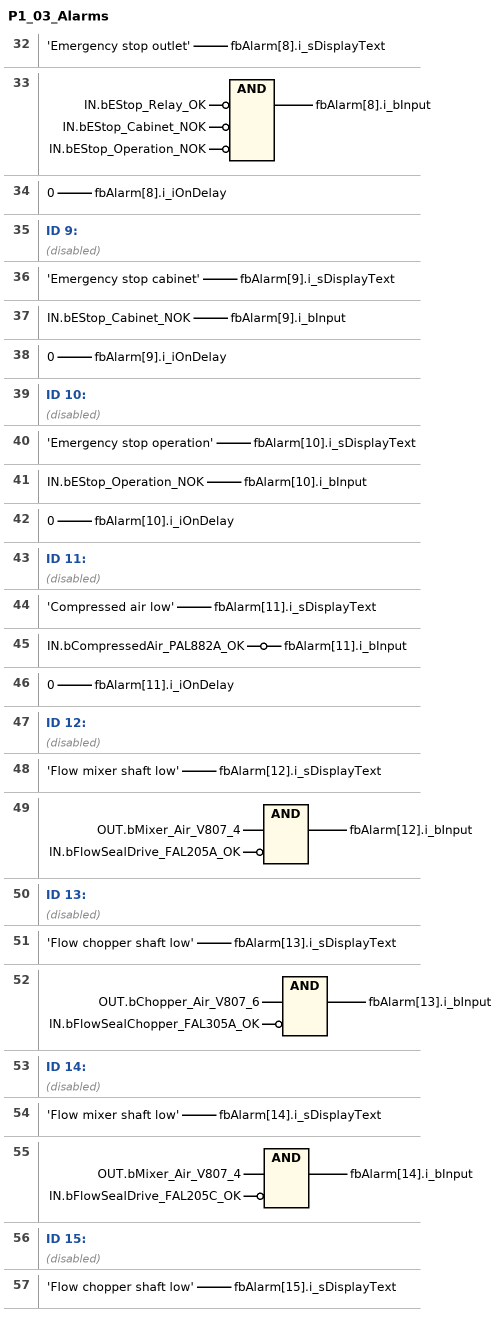
// NETWORK 32
fbAlarm[8].i_sDisplayText := 'Emergency stop outlet';

// NETWORK 33
fbAlarm[8].i_bInput := NOT IN.bEStop_Relay_OK AND NOT IN.bEStop_Cabinet_NOK AND NOT IN.bEStop_Operation_NOK;

// NETWORK 34
fbAlarm[8].i_iOnDelay := 0;

// NETWORK 35 (disabled)
// label: ID 9

// NETWORK 36
fbAlarm[9].i_sDisplayText := 'Emergency stop cabinet';

// NETWORK 37
fbAlarm[9].i_bInput := IN.bEStop_Cabinet_NOK;

// NETWORK 38
fbAlarm[9].i_iOnDelay := 0;

// NETWORK 39 (disabled)
// label: ID 10

// NETWORK 40
fbAlarm[10].i_sDisplayText := 'Emergency stop operation';

// NETWORK 41
fbAlarm[10].i_bInput := IN.bEStop_Operation_NOK;

// NETWORK 42
fbAlarm[10].i_iOnDelay := 0;

// NETWORK 43 (disabled)
// label: ID 11

// NETWORK 44
fbAlarm[11].i_sDisplayText := 'Compressed air low';

// NETWORK 45
fbAlarm[11].i_bInput := NOT IN.bCompressedAir_PAL882A_OK;

// NETWORK 46
fbAlarm[11].i_iOnDelay := 0;

// NETWORK 47 (disabled)
// label: ID 12

// NETWORK 48
fbAlarm[12].i_sDisplayText := 'Flow mixer shaft low';

// NETWORK 49
fbAlarm[12].i_bInput := OUT.bMixer_Air_V807_4 AND NOT IN.bFlowSealDrive_FAL205A_OK;

// NETWORK 50 (disabled)
// label: ID 13

// NETWORK 51
fbAlarm[13].i_sDisplayText := 'Flow chopper shaft low';

// NETWORK 52
fbAlarm[13].i_bInput := OUT.bChopper_Air_V807_6 AND NOT IN.bFlowSealChopper_FAL305A_OK;

// NETWORK 53 (disabled)
// label: ID 14

// NETWORK 54
fbAlarm[14].i_sDisplayText := 'Flow mixer shaft low';

// NETWORK 55
fbAlarm[14].i_bInput := OUT.bMixer_Air_V807_4 AND NOT IN.bFlowSealDrive_FAL205C_OK;

// NETWORK 56 (disabled)
// label: ID 15

// NETWORK 57
fbAlarm[15].i_sDisplayText := 'Flow chopper shaft low';

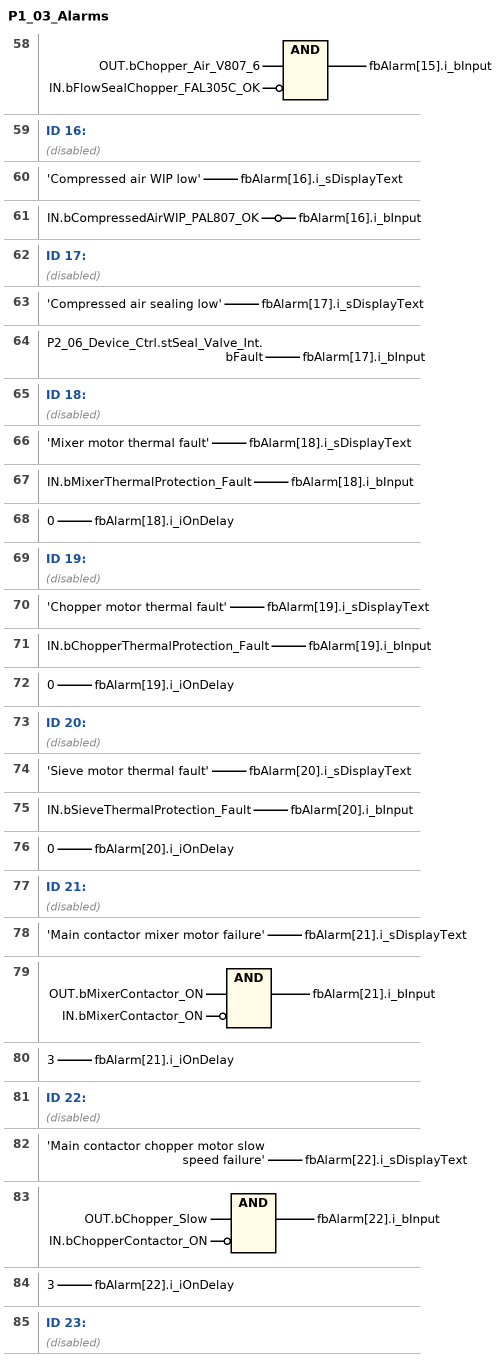
// NETWORK 58
fbAlarm[15].i_bInput := OUT.bChopper_Air_V807_6 AND NOT IN.bFlowSealChopper_FAL305C_OK;

// NETWORK 59 (disabled)
// label: ID 16

// NETWORK 60
fbAlarm[16].i_sDisplayText := 'Compressed air WIP low';

// NETWORK 61
fbAlarm[16].i_bInput := NOT IN.bCompressedAirWIP_PAL807_OK;

// NETWORK 62 (disabled)
// label: ID 17

// NETWORK 63
fbAlarm[17].i_sDisplayText := 'Compressed air sealing low';

// NETWORK 64
fbAlarm[17].i_bInput := P2_06_Device_Ctrl.stSeal_Valve_Int.bFault;

// NETWORK 65 (disabled)
// label: ID 18

// NETWORK 66
fbAlarm[18].i_sDisplayText := 'Mixer motor thermal fault';

// NETWORK 67
fbAlarm[18].i_bInput := IN.bMixerThermalProtection_Fault;

// NETWORK 68
fbAlarm[18].i_iOnDelay := 0;

// NETWORK 69 (disabled)
// label: ID 19

// NETWORK 70
fbAlarm[19].i_sDisplayText := 'Chopper motor thermal fault';

// NETWORK 71
fbAlarm[19].i_bInput := IN.bChopperThermalProtection_Fault;

// NETWORK 72
fbAlarm[19].i_iOnDelay := 0;

// NETWORK 73 (disabled)
// label: ID 20

// NETWORK 74
fbAlarm[20].i_sDisplayText := 'Sieve motor thermal fault';

// NETWORK 75
fbAlarm[20].i_bInput := IN.bSieveThermalProtection_Fault;

// NETWORK 76
fbAlarm[20].i_iOnDelay := 0;

// NETWORK 77 (disabled)
// label: ID 21

// NETWORK 78
fbAlarm[21].i_sDisplayText := 'Main contactor mixer motor failure';

// NETWORK 79
fbAlarm[21].i_bInput := OUT.bMixerContactor_ON AND NOT IN.bMixerContactor_ON;

// NETWORK 80
fbAlarm[21].i_iOnDelay := 3;

// NETWORK 81 (disabled)
// label: ID 22

// NETWORK 82
fbAlarm[22].i_sDisplayText := 'Main contactor chopper motor slow speed failure';

// NETWORK 83
fbAlarm[22].i_bInput := OUT.bChopper_Slow AND NOT IN.bChopperContactor_ON;

// NETWORK 84
fbAlarm[22].i_iOnDelay := 3;

// NETWORK 85 (disabled)
// label: ID 23

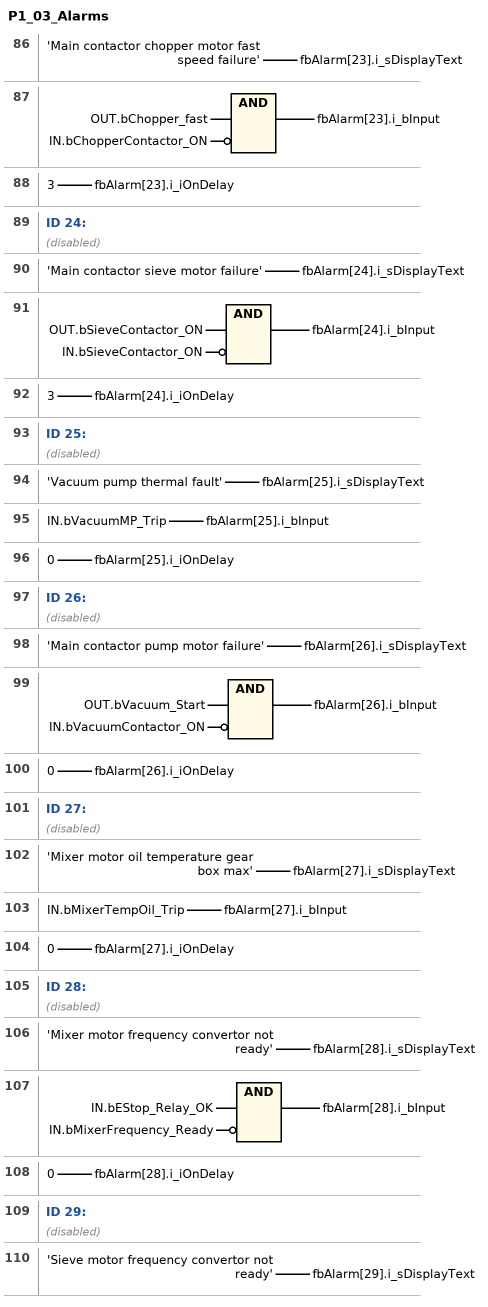
// NETWORK 86
fbAlarm[23].i_sDisplayText := 'Main contactor chopper motor fast speed failure';

// NETWORK 87
fbAlarm[23].i_bInput := OUT.bChopper_fast AND NOT IN.bChopperContactor_ON;

// NETWORK 88
fbAlarm[23].i_iOnDelay := 3;

// NETWORK 89 (disabled)
// label: ID 24

// NETWORK 90
fbAlarm[24].i_sDisplayText := 'Main contactor sieve motor failure';

// NETWORK 91
fbAlarm[24].i_bInput := OUT.bSieveContactor_ON AND NOT IN.bSieveContactor_ON;

// NETWORK 92
fbAlarm[24].i_iOnDelay := 3;

// NETWORK 93 (disabled)
// label: ID 25

// NETWORK 94
fbAlarm[25].i_sDisplayText := 'Vacuum pump thermal fault';

// NETWORK 95
fbAlarm[25].i_bInput := IN.bVacuumMP_Trip;

// NETWORK 96
fbAlarm[25].i_iOnDelay := 0;

// NETWORK 97 (disabled)
// label: ID 26

// NETWORK 98
fbAlarm[26].i_sDisplayText := 'Main contactor pump motor failure';

// NETWORK 99
fbAlarm[26].i_bInput := OUT.bVacuum_Start AND NOT IN.bVacuumContactor_ON;

// NETWORK 100
fbAlarm[26].i_iOnDelay := 0;

// NETWORK 101 (disabled)
// label: ID 27

// NETWORK 102
fbAlarm[27].i_sDisplayText := 'Mixer motor oil temperature gear box max';

// NETWORK 103
fbAlarm[27].i_bInput := IN.bMixerTempOil_Trip;

// NETWORK 104
fbAlarm[27].i_iOnDelay := 0;

// NETWORK 105 (disabled)
// label: ID 28

// NETWORK 106
fbAlarm[28].i_sDisplayText := 'Mixer motor frequency convertor not ready';

// NETWORK 107
fbAlarm[28].i_bInput := IN.bEStop_Relay_OK AND NOT IN.bMixerFrequency_Ready;

// NETWORK 108
fbAlarm[28].i_iOnDelay := 0;

// NETWORK 109 (disabled)
// label: ID 29

// NETWORK 110
fbAlarm[29].i_sDisplayText := 'Sieve motor frequency convertor not ready';

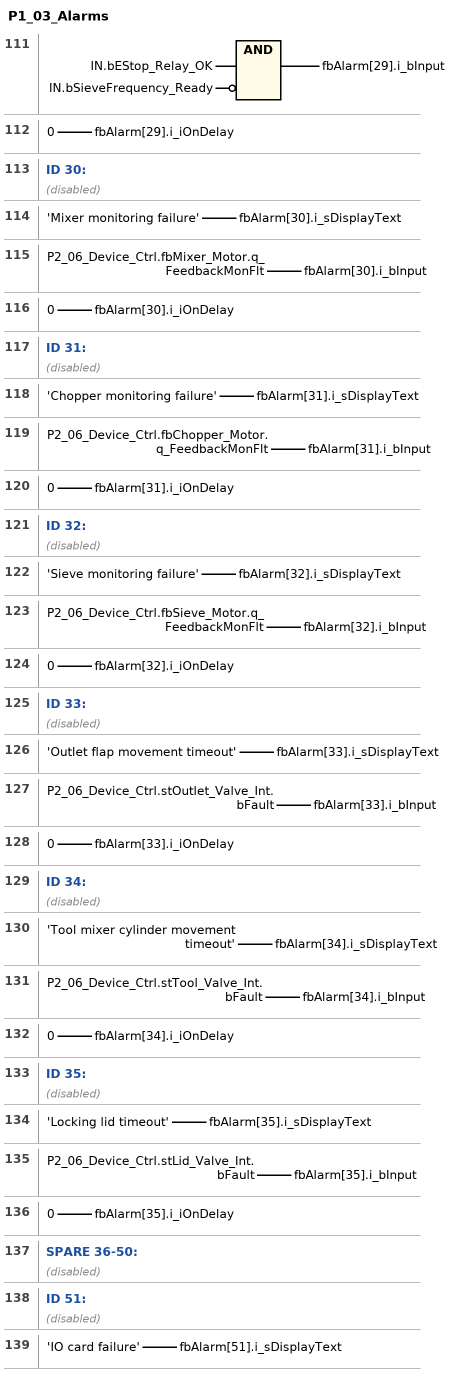
// NETWORK 111
fbAlarm[29].i_bInput := IN.bEStop_Relay_OK AND NOT IN.bSieveFrequency_Ready;

// NETWORK 112
fbAlarm[29].i_iOnDelay := 0;

// NETWORK 113 (disabled)
// label: ID 30

// NETWORK 114
fbAlarm[30].i_sDisplayText := 'Mixer monitoring failure';

// NETWORK 115
fbAlarm[30].i_bInput := P2_06_Device_Ctrl.fbMixer_Motor.q_FeedbackMonFlt;

// NETWORK 116
fbAlarm[30].i_iOnDelay := 0;

// NETWORK 117 (disabled)
// label: ID 31

// NETWORK 118
fbAlarm[31].i_sDisplayText := 'Chopper monitoring failure';

// NETWORK 119
fbAlarm[31].i_bInput := P2_06_Device_Ctrl.fbChopper_Motor.q_FeedbackMonFlt;

// NETWORK 120
fbAlarm[31].i_iOnDelay := 0;

// NETWORK 121 (disabled)
// label: ID 32

// NETWORK 122
fbAlarm[32].i_sDisplayText := 'Sieve monitoring failure';

// NETWORK 123
fbAlarm[32].i_bInput := P2_06_Device_Ctrl.fbSieve_Motor.q_FeedbackMonFlt;

// NETWORK 124
fbAlarm[32].i_iOnDelay := 0;

// NETWORK 125 (disabled)
// label: ID 33

// NETWORK 126
fbAlarm[33].i_sDisplayText := 'Outlet flap movement timeout';

// NETWORK 127
fbAlarm[33].i_bInput := P2_06_Device_Ctrl.stOutlet_Valve_Int.bFault;

// NETWORK 128
fbAlarm[33].i_iOnDelay := 0;

// NETWORK 129 (disabled)
// label: ID 34

// NETWORK 130
fbAlarm[34].i_sDisplayText := 'Tool mixer cylinder movement timeout';

// NETWORK 131
fbAlarm[34].i_bInput := P2_06_Device_Ctrl.stTool_Valve_Int.bFault;

// NETWORK 132
fbAlarm[34].i_iOnDelay := 0;

// NETWORK 133 (disabled)
// label: ID 35

// NETWORK 134
fbAlarm[35].i_sDisplayText := 'Locking lid timeout';

// NETWORK 135
fbAlarm[35].i_bInput := P2_06_Device_Ctrl.stLid_Valve_Int.bFault;

// NETWORK 136
fbAlarm[35].i_iOnDelay := 0;

// NETWORK 137 (disabled)
// label: SPARE 36-50

// NETWORK 138 (disabled)
// label: ID 51

// NETWORK 139
fbAlarm[51].i_sDisplayText := 'IO card failure';

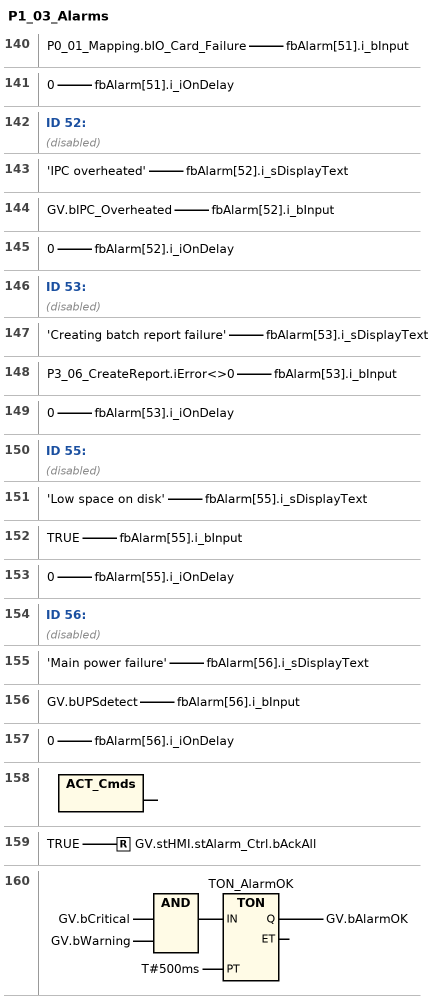
// NETWORK 140
fbAlarm[51].i_bInput := P0_01_Mapping.bIO_Card_Failure;

// NETWORK 141
fbAlarm[51].i_iOnDelay := 0;

// NETWORK 142 (disabled)
// label: ID 52

// NETWORK 143
fbAlarm[52].i_sDisplayText := 'IPC overheated';

// NETWORK 144
fbAlarm[52].i_bInput := GV.bIPC_Overheated;

// NETWORK 145
fbAlarm[52].i_iOnDelay := 0;

// NETWORK 146 (disabled)
// label: ID 53

// NETWORK 147
fbAlarm[53].i_sDisplayText := 'Creating batch report failure';

// NETWORK 148
fbAlarm[53].i_bInput := P3_06_CreateReport.iError<>0;

// NETWORK 149
fbAlarm[53].i_iOnDelay := 0;

// NETWORK 150 (disabled)
// label: ID 55

// NETWORK 151
fbAlarm[55].i_sDisplayText := 'Low space on disk';

// NETWORK 152
fbAlarm[55].i_bInput := TRUE;

// NETWORK 153
fbAlarm[55].i_iOnDelay := 0;

// NETWORK 154 (disabled)
// label: ID 56

// NETWORK 155
fbAlarm[56].i_sDisplayText := 'Main power failure';

// NETWORK 156
fbAlarm[56].i_bInput := GV.bUPSdetect;

// NETWORK 157
fbAlarm[56].i_iOnDelay := 0;

// NETWORK 158
ACT_Cmds();

// NETWORK 159
GV.stHMI.stAlarm_Ctrl.bAckAll R= TRUE;

// NETWORK 160
TON_AlarmOK(IN := GV.bCritical AND GV.bWarning, PT := T#500ms); // TON
GV.bAlarmOK := TON_AlarmOK.Q;

ACTION ACT_Cmds:
GV.bCritical:=TRUE;
GV.bWarning:=TRUE;
bAlarmDisabled:=FALSE;
FOR i:=0 TO 50 DO
	//Init Function blocks
	fbAlarm[i](i_iID:=i,
			   i_bActive:=GV.stAlarm.Active[i],
			   q_bActive=>GV.stAlarm.Raise[i]);			
			   
	fbAlarm[i].i_bEnable:=TRUE;
	IF GV.stAlarm.Active[i] THEN
		IF i <= 25 THEN
			GV.bCritical:=FALSE;
		ELSIF i > 25 THEN
			GV.bWarning:=FALSE;
		END_IF
	END_IF
	
	//Raise
	IF GV.stAlarm.Raise[i] THEN
		GV.stAlarm.Alarm[i].Raise(0);
	END_IF
	
	//Active
	GV.stAlarm.Active[i]:=GV.stAlarm.Alarm[i].bActive;
	
	//Ack
	IF GV.stAlarm.Alarm[i].eConfirmationState = 3 OR GV.stHMI.stAlarm_Ctrl.bAckAll THEN
		GV.stAlarm.Alarm[i].Clear(0,1);
	END_IF
	
	//Clear warnings 
	IF GV.stAlarm.Active[i] AND NOT fbAlarm[i].i_bInput AND i>=25 THEN
		GV.stAlarm.Alarm[i].Clear(0,1);
	END_IF
	
	//Check disabled
	IF NOT fbAlarm[i].i_bEnable THEN
		bAlarmDisabled:=TRUE;
	END_IF
END_FOR
END_ACTION

ACTION ACT_Init:
IF MAIN.bFirstCycle THEN
	//Critical
	GV.stAlarm.Alarm[1].CreateEx(TC_EVENTS.Alarms.AlarmsEvent1,1,0);
	GV.stAlarm.Alarm[2].CreateEx(TC_EVENTS.Alarms.AlarmsEvent2,1,0);
	GV.stAlarm.Alarm[3].CreateEx(TC_EVENTS.Alarms.AlarmsEvent3,1,0);
	GV.stAlarm.Alarm[4].CreateEx(TC_EVENTS.Alarms.AlarmsEvent4,1,0);
	GV.stAlarm.Alarm[5].CreateEx(TC_EVENTS.Alarms.AlarmsEvent5,1,0);
	GV.stAlarm.Alarm[6].CreateEx(TC_EVENTS.Alarms.AlarmsEvent6,1,0);
	GV.stAlarm.Alarm[7].CreateEx(TC_EVENTS.Alarms.AlarmsEvent7,1,0);
	GV.stAlarm.Alarm[8].CreateEx(TC_EVENTS.Alarms.AlarmsEvent8,1,0);
	GV.stAlarm.Alarm[9].CreateEx(TC_EVENTS.Alarms.AlarmsEvent9,1,0);
	GV.stAlarm.Alarm[10].CreateEx(TC_EVENTS.Alarms.AlarmsEvent10,1,0);
	GV.stAlarm.Alarm[11].CreateEx(TC_EVENTS.Alarms.AlarmsEvent11,1,0);
	GV.stAlarm.Alarm[12].CreateEx(TC_EVENTS.Alarms.AlarmsEvent12,1,0);
	GV.stAlarm.Alarm[13].CreateEx(TC_EVENTS.Alarms.AlarmsEvent13,1,0);
	GV.stAlarm.Alarm[14].CreateEx(TC_EVENTS.Alarms.AlarmsEvent14,1,0);
	GV.stAlarm.Alarm[15].CreateEx(TC_EVENTS.Alarms.AlarmsEvent15,1,0);
	GV.stAlarm.Alarm[16].CreateEx(TC_EVENTS.Alarms.AlarmsEvent16,1,0);
	GV.stAlarm.Alarm[17].CreateEx(TC_EVENTS.Alarms.AlarmsEvent17,1,0);
	GV.stAlarm.Alarm[18].CreateEx(TC_EVENTS.Alarms.AlarmsEvent18,1,0);
	GV.stAlarm.Alarm[19].CreateEx(TC_EVENTS.Alarms.AlarmsEvent19,1,0);
	GV.stAlarm.Alarm[20].CreateEx(TC_EVENTS.Alarms.AlarmsEvent20,1,0);
	GV.stAlarm.Alarm[21].CreateEx(TC_EVENTS.Alarms.AlarmsEvent21,1,0);
	GV.stAlarm.Alarm[22].CreateEx(TC_EVENTS.Alarms.AlarmsEvent22,1,0);
	GV.stAlarm.Alarm[23].CreateEx(TC_EVENTS.Alarms.AlarmsEvent23,1,0);
	GV.stAlarm.Alarm[24].CreateEx(TC_EVENTS.Alarms.AlarmsEvent24,1,0);
	GV.stAlarm.Alarm[25].CreateEx(TC_EVENTS.Alarms.AlarmsEvent25,1,0);
	GV.stAlarm.Alarm[26].CreateEx(TC_EVENTS.Alarms.AlarmsEvent26,1,0);
	GV.stAlarm.Alarm[27].CreateEx(TC_EVENTS.Alarms.AlarmsEvent27,1,0);
	GV.stAlarm.Alarm[28].CreateEx(TC_EVENTS.Alarms.AlarmsEvent28,1,0);
	GV.stAlarm.Alarm[29].CreateEx(TC_EVENTS.Alarms.AlarmsEvent29,1,0);
	GV.stAlarm.Alarm[30].CreateEx(TC_EVENTS.Alarms.AlarmsEvent30,1,0);
	GV.stAlarm.Alarm[31].CreateEx(TC_EVENTS.Alarms.AlarmsEvent31,1,0);
	GV.stAlarm.Alarm[32].CreateEx(TC_EVENTS.Alarms.AlarmsEvent32,1,0);
	GV.stAlarm.Alarm[33].CreateEx(TC_EVENTS.Alarms.AlarmsEvent33,1,0);
	GV.stAlarm.Alarm[34].CreateEx(TC_EVENTS.Alarms.AlarmsEvent34,1,0);
	GV.stAlarm.Alarm[35].CreateEx(TC_EVENTS.Alarms.AlarmsEvent35,1,0);
	GV.stAlarm.Alarm[36].CreateEx(TC_EVENTS.Alarms.AlarmsEvent36,1,0);
	GV.stAlarm.Alarm[37].CreateEx(TC_EVENTS.Alarms.AlarmsEvent37,1,0);
	GV.stAlarm.Alarm[38].CreateEx(TC_EVENTS.Alarms.AlarmsEvent38,1,0);
	GV.stAlarm.Alarm[39].CreateEx(TC_EVENTS.Alarms.AlarmsEvent39,1,0);
	GV.stAlarm.Alarm[40].CreateEx(TC_EVENTS.Alarms.AlarmsEvent40,1,0);	
	GV.stAlarm.Alarm[41].CreateEx(TC_EVENTS.Alarms.AlarmsEvent41,1,0);
	GV.stAlarm.Alarm[42].CreateEx(TC_EVENTS.Alarms.AlarmsEvent42,1,0);
	GV.stAlarm.Alarm[43].CreateEx(TC_EVENTS.Alarms.AlarmsEvent43,1,0);
	GV.stAlarm.Alarm[44].CreateEx(TC_EVENTS.Alarms.AlarmsEvent44,1,0);
	GV.stAlarm.Alarm[45].CreateEx(TC_EVENTS.Alarms.AlarmsEvent45,1,0);
	GV.stAlarm.Alarm[46].CreateEx(TC_EVENTS.Alarms.AlarmsEvent46,1,0);
	GV.stAlarm.Alarm[47].CreateEx(TC_EVENTS.Alarms.AlarmsEvent47,1,0);
	GV.stAlarm.Alarm[48].CreateEx(TC_EVENTS.Alarms.AlarmsEvent48,1,0);
	GV.stAlarm.Alarm[49].CreateEx(TC_EVENTS.Alarms.AlarmsEvent49,1,0);
	GV.stAlarm.Alarm[50].CreateEx(TC_EVENTS.Alarms.AlarmsEvent50,1,0);
	GV.stAlarm.Alarm[51].CreateEx(TC_EVENTS.Alarms.AlarmsEvent51,1,0);
	GV.stAlarm.Alarm[52].CreateEx(TC_EVENTS.Alarms.AlarmsEvent52,1,0);
	GV.stAlarm.Alarm[53].CreateEx(TC_EVENTS.Alarms.AlarmsEvent53,1,0);
	GV.stAlarm.Alarm[54].CreateEx(TC_EVENTS.Alarms.AlarmsEvent54,1,0);
	GV.stAlarm.Alarm[55].CreateEx(TC_EVENTS.Alarms.AlarmsEvent55,1,0);
	GV.stAlarm.Alarm[56].CreateEx(TC_EVENTS.Alarms.AlarmsEvent56,1,0);
	GV.stAlarm.Alarm[57].CreateEx(TC_EVENTS.Alarms.AlarmsEvent57,1,0);
	GV.stAlarm.Alarm[58].CreateEx(TC_EVENTS.Alarms.AlarmsEvent58,1,0);
	GV.stAlarm.Alarm[59].CreateEx(TC_EVENTS.Alarms.AlarmsEvent59,1,0);
	GV.stAlarm.Alarm[60].CreateEx(TC_EVENTS.Alarms.AlarmsEvent60,1,0);
	//SP
	GV.stAlarm.Alarm[61].CreateEx(TC_EVENTS.Alarms.AlarmsEvent61,1,0);
	GV.stAlarm.Alarm[62].CreateEx(TC_EVENTS.Alarms.AlarmsEvent62,1,0);
	GV.stAlarm.Alarm[63].CreateEx(TC_EVENTS.Alarms.AlarmsEvent63,1,0);
	GV.stAlarm.Alarm[64].CreateEx(TC_EVENTS.Alarms.AlarmsEvent64,1,0);
	GV.stAlarm.Alarm[65].CreateEx(TC_EVENTS.Alarms.AlarmsEvent65,1,0);
	GV.stAlarm.Alarm[66].CreateEx(TC_EVENTS.Alarms.AlarmsEvent66,1,0);
	GV.stAlarm.Alarm[67].CreateEx(TC_EVENTS.Alarms.AlarmsEvent67,1,0);
	GV.stAlarm.Alarm[68].CreateEx(TC_EVENTS.Alarms.AlarmsEvent68,1,0);
	GV.stAlarm.Alarm[69].CreateEx(TC_EVENTS.Alarms.AlarmsEvent69,1,0);
	GV.stAlarm.Alarm[70].CreateEx(TC_EVENTS.Alarms.AlarmsEvent70,1,0);
END_IF
END_ACTION

END_PROGRAM

// ---- FBs/FB_AlarmDiagnostic.TcPOU
FUNCTION_BLOCK FB_AlarmDiagnostic
VAR_INPUT
	i_bEnable				:BOOL:=TRUE;
	i_iID					:INT;
	i_bInput				:BOOL;
	i_iOnDelay				:INT;
	i_bReset				:BOOL;
	i_bTest					:BOOL;
	i_bActive				:BOOL;
END_VAR
VAR_OUTPUT
	q_bActive				:BOOL;
	q_iDetections			:INT;
END_VAR
VAR
	TON						:TON;
END_VAR
VAR // added by the converter: edge detectors and wires of the graphical bodies
    _rt1 : R_TRIG;
    _w1 : BOOL;
END_VAR

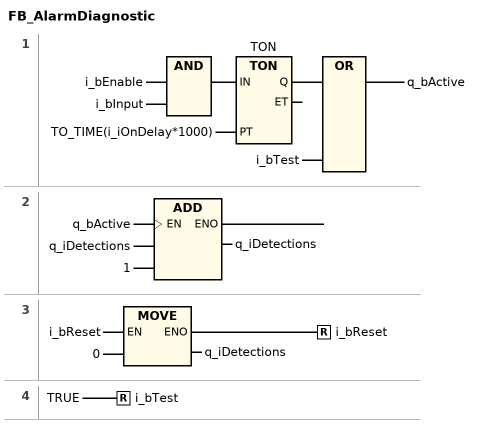
// NETWORK 1
TON(IN := i_bEnable AND i_bInput, PT := TO_TIME(i_iOnDelay*1000));
q_bActive := TON.Q OR i_bTest;

// NETWORK 2
_rt1(CLK := q_bActive);
IF _rt1.Q THEN q_iDetections := q_iDetections + 1; END_IF

// NETWORK 3
_w1 := i_bReset;
IF _w1 THEN q_iDetections := 0; END_IF
i_bReset R= _w1;

// NETWORK 4
i_bTest R= TRUE;

END_FUNCTION_BLOCK

// ---- POUs/2. Process/P2_06_Device_Ctrl.TcPOU
PROGRAM P2_06_Device_Ctrl
VAR
	fbMixer_Motor					:FB_MotorFreqCtrl;
	fbMixerMotor_Speed				:FB_AnalogOutput_v01;
	fbSieve_Motor					:FB_MotorFreqCtrl;
	fbSieveMotor_Speed				:FB_AnalogOutput_v01;
	fbChopper_Motor					:FB_MotorCoilsCtrl;
	fbPump_Motor					:FB_CoilCtrl;
	
	fbSP_Temperature_PID			:FB_PID;
	
	fbSP_Mixer_Motor				:FB_MotorFreqCtrl;
	fbSP_MixerMotor_Speed			:FB_AnalogOutput_v01;
	fbSP_Pressure					:FB_AnalogOutput_v02;
	
	fbOutlet_Valve					:FB_ValveCtrl52;
	fbLid_Valve						:FB_ValveCtrl52;
	fbSieveSeal_Valve				:FB_ValveCtrl52;
	fbPurge_Valve					:FB_ValveCtrl52;
	fbTool_Valve					:FB_ValveCtrl52;
	
	fbCleaningAir_Valve				:FB_ValveCtrl32;
	fbPurifiedWater_Valve			:FB_ValveCtrl32;
	fbWarmWater_Valve				:FB_ValveCtrl32;
	fbColdWater_Valve				:FB_ValveCtrl32;
	fbMixerWIP_Valve				:FB_ValveCtrl32;
	fbChopperWIP_Valve				:FB_ValveCtrl32;
	fbSPWIP_Valve					:FB_ValveCtrl32;
	fbSPWIPDrain_Valve				:FB_ValveCtrl32;
	fbMainDrain_Valve				:FB_ValveCtrl32;
	
	fbAspiration_Valve				:FB_ValveCtrl32;
	fbVacuum_Valve					:FB_ValveCtrl32;
	fbFilterClean_Valve				:FB_ValveCtrl32;
	fbAirSeal_Valve					:FB_ValveCtrl32;
	fbMixerAir_Valve				:FB_ValveCtrl32;
	fbChopperAir_Valve				:FB_ValveCtrl32;
	
	
	
	

END_VAR

VAR PERSISTENT
	stMixer_Motor_Int				:ST_Interface_MotorCtrl;
	stSieve_Motor_Int				:ST_Interface_MotorCtrl;
	stChopper_Motor_Int				:ST_Interface_MotorCoilsCtrl;
	stPump_Motor_Int				:ST_Interface_CoilCtrl;
	
	stSP_Mixer_Motor_Int			:ST_Interface_MotorCtrl;
	stSP_Temperature_Int			:ST_Interface_PidCtrl;
	
	stOutlet_Valve_Int				:ST_Interface_ValveCtrl;
	stLid_Valve_Int					:ST_Interface_ValveCtrl;
	stSeal_Valve_Int				:ST_Interface_ValveCtrl;
	stPurge_Valve_Int				:ST_Interface_ValveCtrl;
	stTool_Valve_Int				:ST_Interface_ValveCtrl;
	
	stCleaningAir_Valve_INT			:ST_Interface_ValveCtrl;
	stPurifiedWater_Valve_INT		:ST_Interface_ValveCtrl;
	stWarmWater_Valve_Int			:ST_Interface_ValveCtrl;
	stColdWater_Valve_Int			:ST_Interface_ValveCtrl;
	stMixerWIP_Valve_Int			:ST_Interface_ValveCtrl;
	stChopperWIP_Valve_Int			:ST_Interface_ValveCtrl;
	stSPWIP_Valve_Int				:ST_Interface_ValveCtrl;
	stSPWIPDrain_Valve_Int			:ST_Interface_ValveCtrl;
	stMainDrain_Valve_Int			:ST_Interface_ValveCtrl;
	
	stAspiration_Valve_Int			:ST_Interface_ValveCtrl;
	stVacuum_Valve_Int				:ST_Interface_ValveCtrl;
	stFilterClean_Valve_Int			:ST_Interface_ValveCtrl;
	stAirSeal_Valve_Int				:ST_Interface_ValveCtrl;
	stMixerAir_Valve_Int			:ST_Interface_ValveCtrl;
	stChopperAir_Valve_Int			:ST_Interface_ValveCtrl;
END_VAR
VAR // added by the converter: edge detectors and wires of the graphical bodies
    _w1, _w2, _w3, _w4, _w5, _w6, _w7, _w8, _w9, _w10 : BOOL;
    _rt1, _rt2 : R_TRIG;
END_VAR

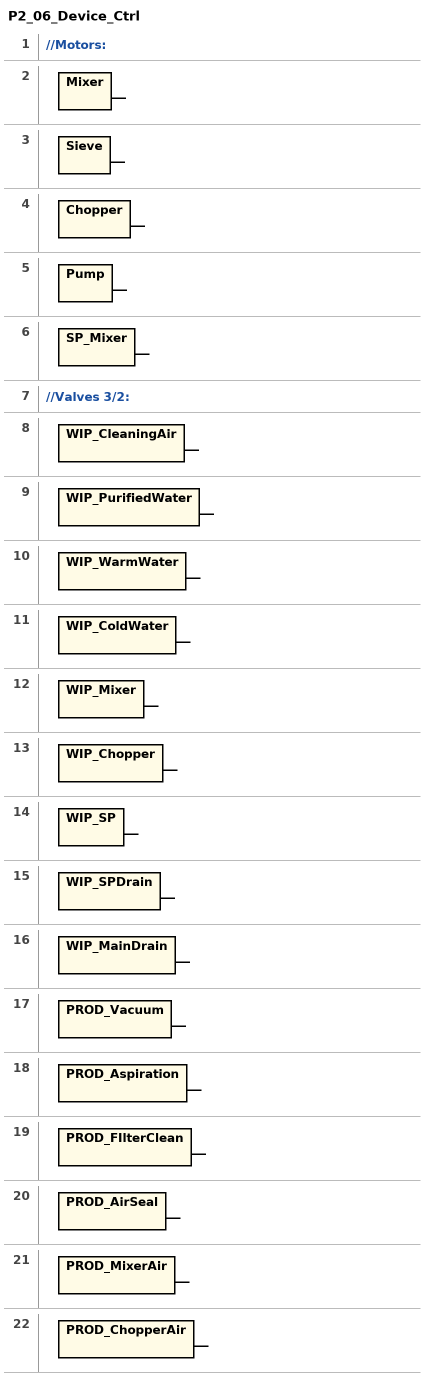
// NETWORK 1
// label: //Motors

// NETWORK 2
Mixer();

// NETWORK 3
Sieve();

// NETWORK 4
Chopper();

// NETWORK 5
Pump();

// NETWORK 6
SP_Mixer();

// NETWORK 7
// label: //Valves 3/2

// NETWORK 8
WIP_CleaningAir();

// NETWORK 9
WIP_PurifiedWater();

// NETWORK 10
WIP_WarmWater();

// NETWORK 11
WIP_ColdWater();

// NETWORK 12
WIP_Mixer();

// NETWORK 13
WIP_Chopper();

// NETWORK 14
WIP_SP();

// NETWORK 15
WIP_SPDrain();

// NETWORK 16
WIP_MainDrain();

// NETWORK 17
PROD_Vacuum();

// NETWORK 18
PROD_Aspiration();

// NETWORK 19
PROD_FIlterClean();

// NETWORK 20
PROD_AirSeal();

// NETWORK 21
PROD_MixerAir();

// NETWORK 22
PROD_ChopperAir();

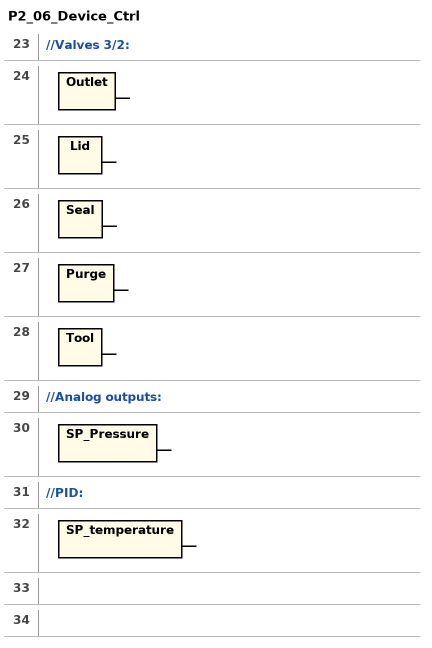
// NETWORK 23
// label: //Valves 3/2

// NETWORK 24
Outlet();

// NETWORK 25
Lid();

// NETWORK 26
Seal();

// NETWORK 27
Purge();

// NETWORK 28
Tool();

// NETWORK 29
// label: //Analog outputs

// NETWORK 30
SP_Pressure();

// NETWORK 31
// label: //PID

// NETWORK 32
SP_temperature();

// NETWORK 33

// NETWORK 34

ACTION Chopper:
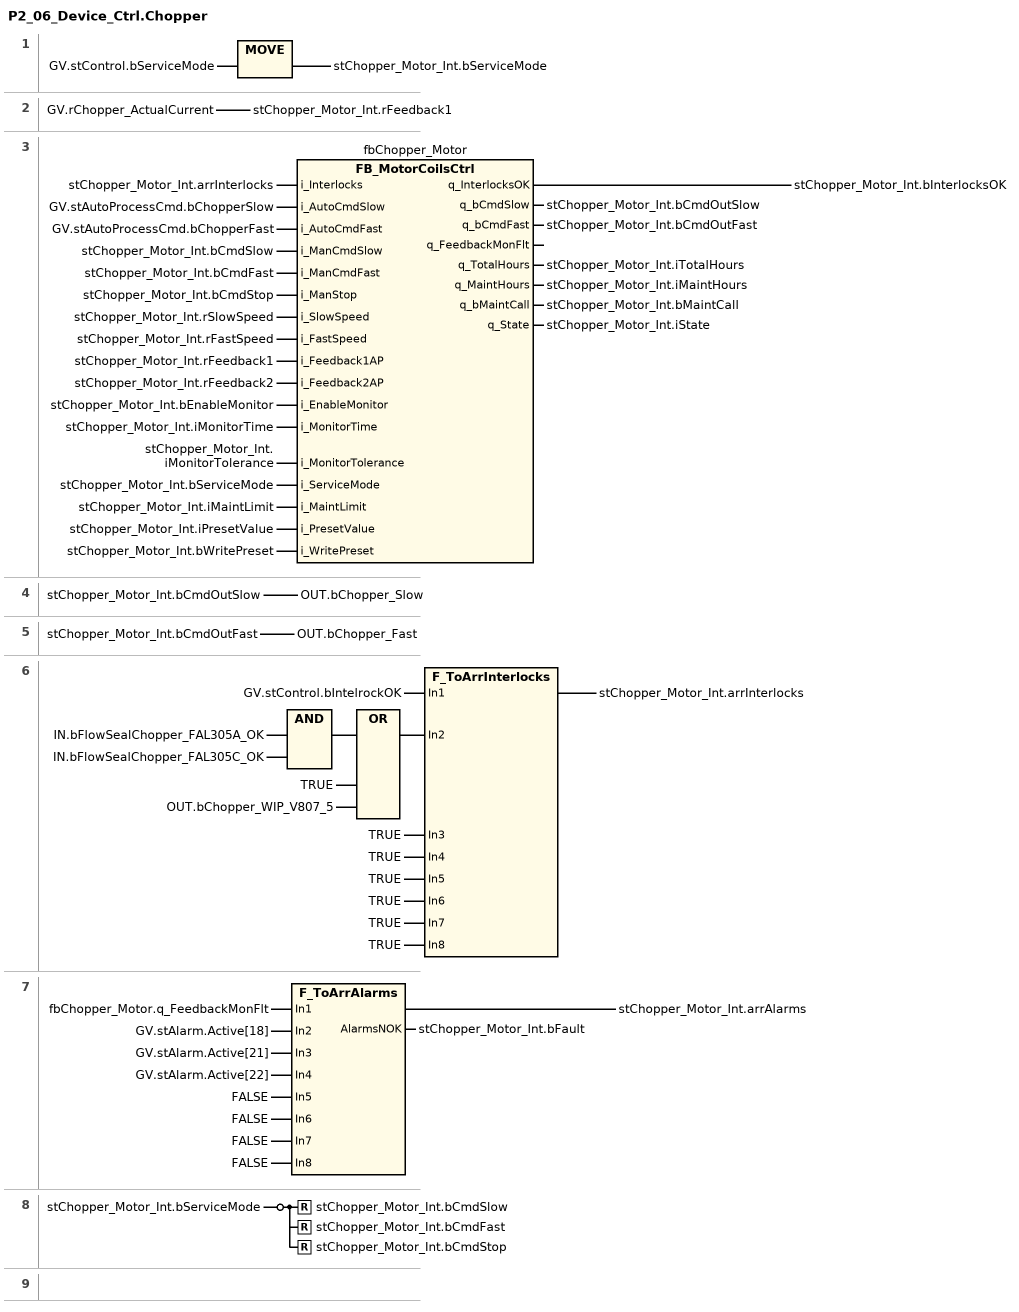
// NETWORK 1
stChopper_Motor_Int.bServiceMode := GV.stControl.bServiceMode;

// NETWORK 2
stChopper_Motor_Int.rFeedback1 := GV.rChopper_ActualCurrent;

// NETWORK 3
fbChopper_Motor(
    i_Interlocks := stChopper_Motor_Int.arrInterlocks,
    i_AutoCmdSlow := GV.stAutoProcessCmd.bChopperSlow,
    i_AutoCmdFast := GV.stAutoProcessCmd.bChopperFast,
    i_ManCmdSlow := stChopper_Motor_Int.bCmdSlow,
    i_ManCmdFast := stChopper_Motor_Int.bCmdFast,
    i_ManStop := stChopper_Motor_Int.bCmdStop,
    i_SlowSpeed := stChopper_Motor_Int.rSlowSpeed,
    i_FastSpeed := stChopper_Motor_Int.rFastSpeed,
    i_Feedback1AP := stChopper_Motor_Int.rFeedback1,
    i_Feedback2AP := stChopper_Motor_Int.rFeedback2,
    i_EnableMonitor := stChopper_Motor_Int.bEnableMonitor,
    i_MonitorTime := stChopper_Motor_Int.iMonitorTime,
    i_MonitorTolerance := stChopper_Motor_Int.iMonitorTolerance,
    i_ServiceMode := stChopper_Motor_Int.bServiceMode,
    i_MaintLimit := stChopper_Motor_Int.iMaintLimit,
    i_PresetValue := stChopper_Motor_Int.iPresetValue,
    i_WritePreset := stChopper_Motor_Int.bWritePreset,
    q_bCmdSlow => stChopper_Motor_Int.bCmdOutSlow,
    q_bCmdFast => stChopper_Motor_Int.bCmdOutFast,
    q_TotalHours => stChopper_Motor_Int.iTotalHours,
    q_MaintHours => stChopper_Motor_Int.iMaintHours,
    q_bMaintCall => stChopper_Motor_Int.bMaintCall,
    q_State => stChopper_Motor_Int.iState); // FB_MotorCoilsCtrl
stChopper_Motor_Int.bInterlocksOK := fbChopper_Motor.q_InterlocksOK;

// NETWORK 4
OUT.bChopper_Slow := stChopper_Motor_Int.bCmdOutSlow;

// NETWORK 5
OUT.bChopper_Fast := stChopper_Motor_Int.bCmdOutFast;

// NETWORK 6
stChopper_Motor_Int.arrInterlocks := F_ToArrInterlocks(In1 := GV.stControl.bIntelrockOK, In2 := IN.bFlowSealChopper_FAL305A_OK AND IN.bFlowSealChopper_FAL305C_OK OR TRUE OR OUT.bChopper_WIP_V807_5, In3 := TRUE, In4 := TRUE, In5 := TRUE, In6 := TRUE, In7 := TRUE, In8 := TRUE);

// NETWORK 7
stChopper_Motor_Int.arrAlarms := F_ToArrAlarms(In1 := fbChopper_Motor.q_FeedbackMonFlt, In2 := GV.stAlarm.Active[18], In3 := GV.stAlarm.Active[21], In4 := GV.stAlarm.Active[22], In5 := FALSE, In6 := FALSE, In7 := FALSE, In8 := FALSE, AlarmsNOK => stChopper_Motor_Int.bFault);

// NETWORK 8
_w1 := NOT stChopper_Motor_Int.bServiceMode;
stChopper_Motor_Int.bCmdSlow R= _w1;
stChopper_Motor_Int.bCmdFast R= _w1;
stChopper_Motor_Int.bCmdStop R= _w1;

// NETWORK 9
END_ACTION

ACTION Lid:
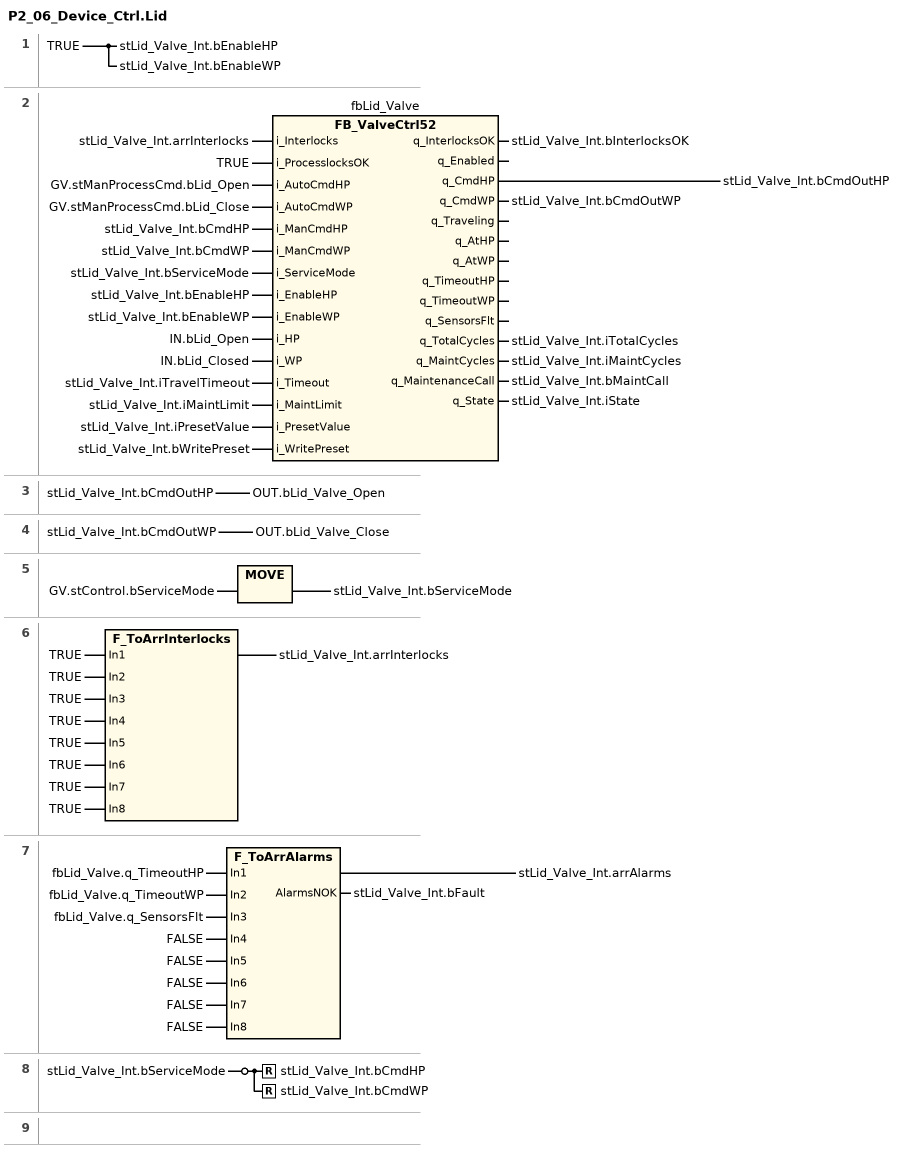
// NETWORK 1
stLid_Valve_Int.bEnableHP := TRUE;
stLid_Valve_Int.bEnableWP := TRUE;

// NETWORK 2
fbLid_Valve(
    i_Interlocks := stLid_Valve_Int.arrInterlocks,
    i_ProcesslocksOK := TRUE,
    i_AutoCmdHP := GV.stManProcessCmd.bLid_Open,
    i_AutoCmdWP := GV.stManProcessCmd.bLid_Close,
    i_ManCmdHP := stLid_Valve_Int.bCmdHP,
    i_ManCmdWP := stLid_Valve_Int.bCmdWP,
    i_ServiceMode := stLid_Valve_Int.bServiceMode,
    i_EnableHP := stLid_Valve_Int.bEnableHP,
    i_EnableWP := stLid_Valve_Int.bEnableWP,
    i_HP := IN.bLid_Open,
    i_WP := IN.bLid_Closed,
    i_Timeout := stLid_Valve_Int.iTravelTimeout,
    i_MaintLimit := stLid_Valve_Int.iMaintLimit,
    i_PresetValue := stLid_Valve_Int.iPresetValue,
    i_WritePreset := stLid_Valve_Int.bWritePreset,
    q_InterlocksOK => stLid_Valve_Int.bInterlocksOK,
    q_CmdWP => stLid_Valve_Int.bCmdOutWP,
    q_TotalCycles => stLid_Valve_Int.iTotalCycles,
    q_MaintCycles => stLid_Valve_Int.iMaintCycles,
    q_MaintenanceCall => stLid_Valve_Int.bMaintCall,
    q_State => stLid_Valve_Int.iState); // FB_ValveCtrl52
stLid_Valve_Int.bCmdOutHP := fbLid_Valve.q_CmdHP;

// NETWORK 3
OUT.bLid_Valve_Open := stLid_Valve_Int.bCmdOutHP;

// NETWORK 4
OUT.bLid_Valve_Close := stLid_Valve_Int.bCmdOutWP;

// NETWORK 5
stLid_Valve_Int.bServiceMode := GV.stControl.bServiceMode;

// NETWORK 6
stLid_Valve_Int.arrInterlocks := F_ToArrInterlocks(In1 := TRUE, In2 := TRUE, In3 := TRUE, In4 := TRUE, In5 := TRUE, In6 := TRUE, In7 := TRUE, In8 := TRUE);

// NETWORK 7
stLid_Valve_Int.arrAlarms := F_ToArrAlarms(In1 := fbLid_Valve.q_TimeoutHP, In2 := fbLid_Valve.q_TimeoutWP, In3 := fbLid_Valve.q_SensorsFlt, In4 := FALSE, In5 := FALSE, In6 := FALSE, In7 := FALSE, In8 := FALSE, AlarmsNOK => stLid_Valve_Int.bFault);

// NETWORK 8
_w2 := NOT stLid_Valve_Int.bServiceMode;
stLid_Valve_Int.bCmdHP R= _w2;
stLid_Valve_Int.bCmdWP R= _w2;

// NETWORK 9
END_ACTION

ACTION Mixer:
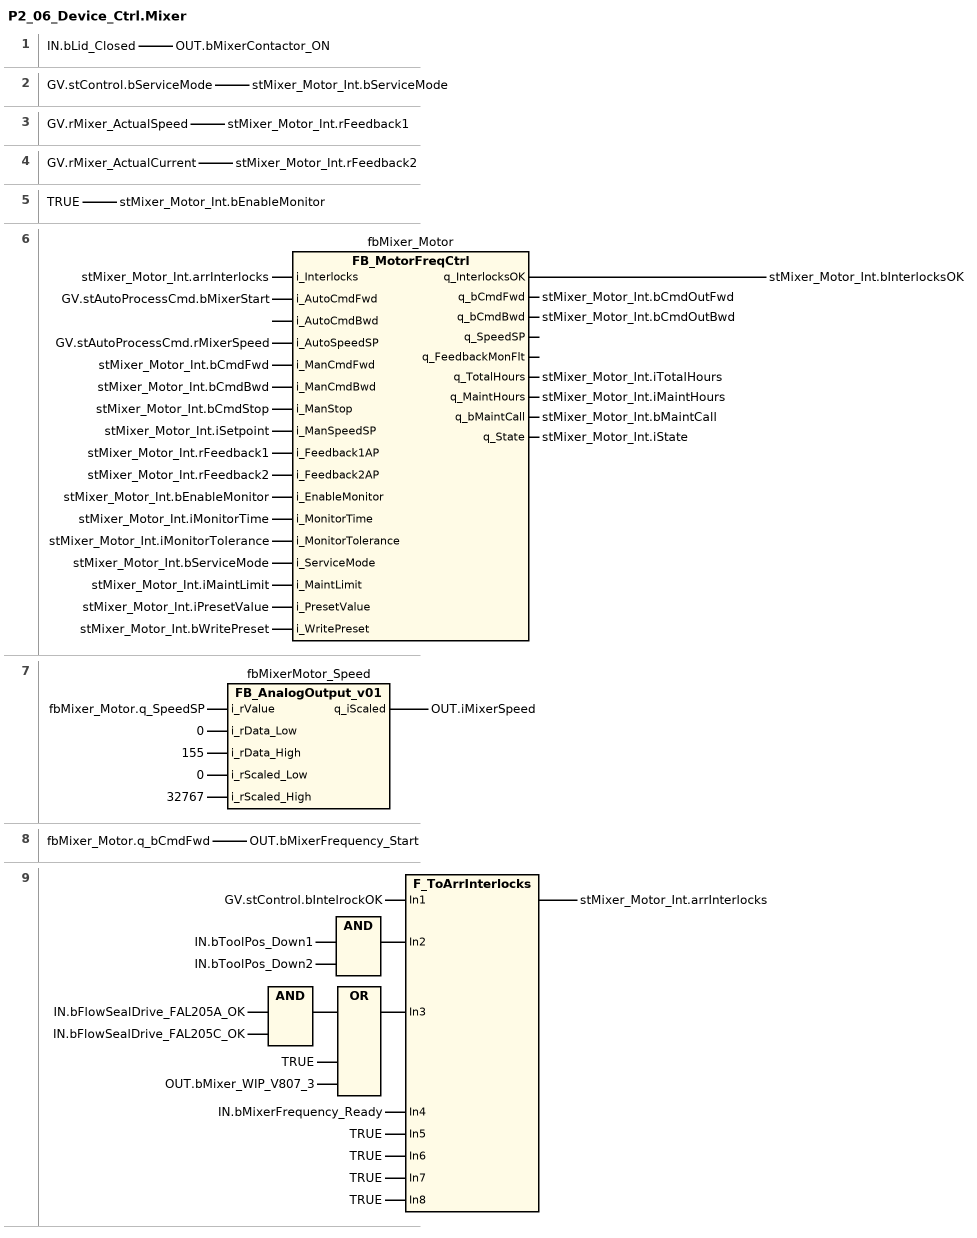
// NETWORK 1
OUT.bMixerContactor_ON := IN.bLid_Closed;

// NETWORK 2
stMixer_Motor_Int.bServiceMode := GV.stControl.bServiceMode;

// NETWORK 3
stMixer_Motor_Int.rFeedback1 := GV.rMixer_ActualSpeed;

// NETWORK 4
stMixer_Motor_Int.rFeedback2 := GV.rMixer_ActualCurrent;

// NETWORK 5
stMixer_Motor_Int.bEnableMonitor := TRUE;

// NETWORK 6
fbMixer_Motor(
    i_Interlocks := stMixer_Motor_Int.arrInterlocks,
    i_AutoCmdFwd := GV.stAutoProcessCmd.bMixerStart,
    i_AutoSpeedSP := GV.stAutoProcessCmd.rMixerSpeed,
    i_ManCmdFwd := stMixer_Motor_Int.bCmdFwd,
    i_ManCmdBwd := stMixer_Motor_Int.bCmdBwd,
    i_ManStop := stMixer_Motor_Int.bCmdStop,
    i_ManSpeedSP := stMixer_Motor_Int.iSetpoint,
    i_Feedback1AP := stMixer_Motor_Int.rFeedback1,
    i_Feedback2AP := stMixer_Motor_Int.rFeedback2,
    i_EnableMonitor := stMixer_Motor_Int.bEnableMonitor,
    i_MonitorTime := stMixer_Motor_Int.iMonitorTime,
    i_MonitorTolerance := stMixer_Motor_Int.iMonitorTolerance,
    i_ServiceMode := stMixer_Motor_Int.bServiceMode,
    i_MaintLimit := stMixer_Motor_Int.iMaintLimit,
    i_PresetValue := stMixer_Motor_Int.iPresetValue,
    i_WritePreset := stMixer_Motor_Int.bWritePreset,
    q_bCmdFwd => stMixer_Motor_Int.bCmdOutFwd,
    q_bCmdBwd => stMixer_Motor_Int.bCmdOutBwd,
    q_TotalHours => stMixer_Motor_Int.iTotalHours,
    q_MaintHours => stMixer_Motor_Int.iMaintHours,
    q_bMaintCall => stMixer_Motor_Int.bMaintCall,
    q_State => stMixer_Motor_Int.iState); // FB_MotorFreqCtrl
stMixer_Motor_Int.bInterlocksOK := fbMixer_Motor.q_InterlocksOK;

// NETWORK 7
fbMixerMotor_Speed(
    i_rValue := fbMixer_Motor.q_SpeedSP,
    i_rData_Low := 0,
    i_rData_High := 155,
    i_rScaled_Low := 0,
    i_rScaled_High := 32767); // FB_AnalogOutput_v01
OUT.iMixerSpeed := fbMixerMotor_Speed.q_iScaled;

// NETWORK 8
OUT.bMixerFrequency_Start := fbMixer_Motor.q_bCmdFwd;

// NETWORK 9
stMixer_Motor_Int.arrInterlocks := F_ToArrInterlocks(In1 := GV.stControl.bIntelrockOK, In2 := IN.bToolPos_Down1 AND IN.bToolPos_Down2, In3 := IN.bFlowSealDrive_FAL205A_OK AND IN.bFlowSealDrive_FAL205C_OK OR TRUE OR OUT.bMixer_WIP_V807_3, In4 := IN.bMixerFrequency_Ready, In5 := TRUE, In6 := TRUE, In7 := TRUE, In8 := TRUE);

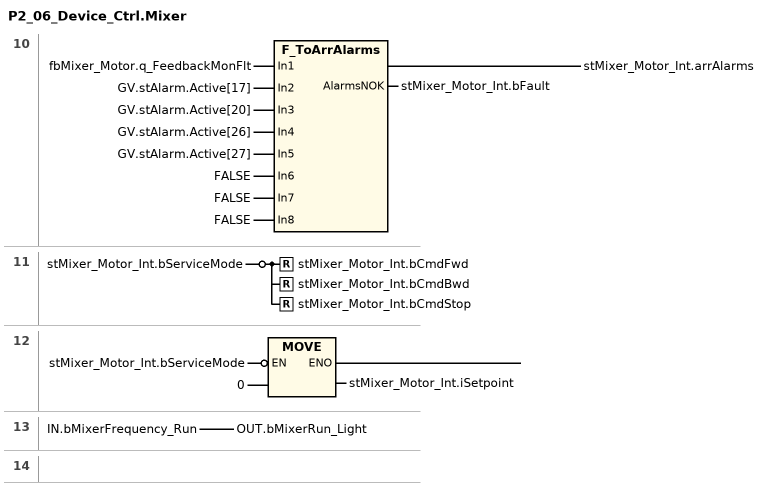
// NETWORK 10
stMixer_Motor_Int.arrAlarms := F_ToArrAlarms(In1 := fbMixer_Motor.q_FeedbackMonFlt, In2 := GV.stAlarm.Active[17], In3 := GV.stAlarm.Active[20], In4 := GV.stAlarm.Active[26], In5 := GV.stAlarm.Active[27], In6 := FALSE, In7 := FALSE, In8 := FALSE, AlarmsNOK => stMixer_Motor_Int.bFault);

// NETWORK 11
_w3 := NOT stMixer_Motor_Int.bServiceMode;
stMixer_Motor_Int.bCmdFwd R= _w3;
stMixer_Motor_Int.bCmdBwd R= _w3;
stMixer_Motor_Int.bCmdStop R= _w3;

// NETWORK 12
IF NOT stMixer_Motor_Int.bServiceMode THEN stMixer_Motor_Int.iSetpoint := 0; END_IF

// NETWORK 13
OUT.bMixerRun_Light := IN.bMixerFrequency_Run;

// NETWORK 14
END_ACTION

ACTION Outlet:
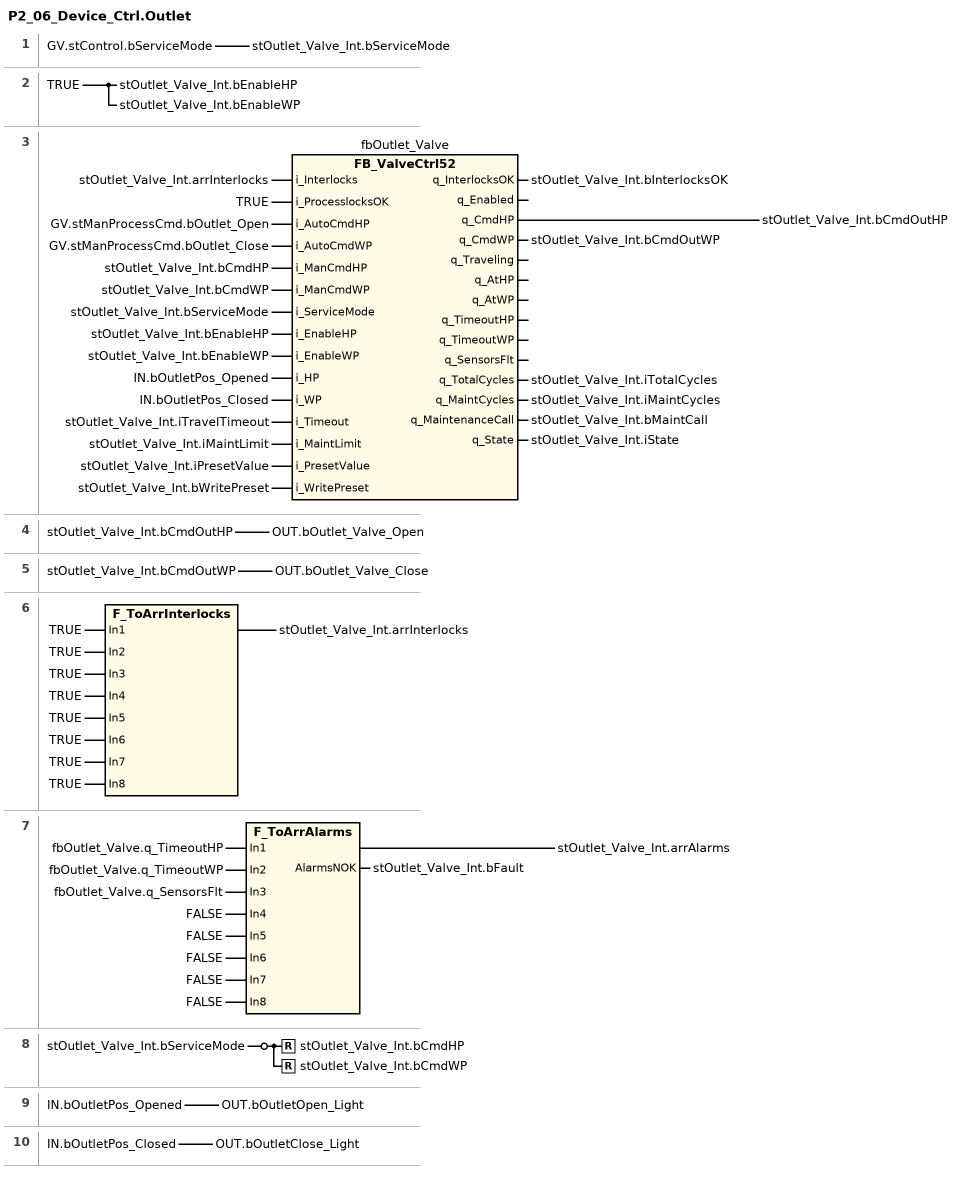
// NETWORK 1
stOutlet_Valve_Int.bServiceMode := GV.stControl.bServiceMode;

// NETWORK 2
stOutlet_Valve_Int.bEnableHP := TRUE;
stOutlet_Valve_Int.bEnableWP := TRUE;

// NETWORK 3
fbOutlet_Valve(
    i_Interlocks := stOutlet_Valve_Int.arrInterlocks,
    i_ProcesslocksOK := TRUE,
    i_AutoCmdHP := GV.stManProcessCmd.bOutlet_Open,
    i_AutoCmdWP := GV.stManProcessCmd.bOutlet_Close,
    i_ManCmdHP := stOutlet_Valve_Int.bCmdHP,
    i_ManCmdWP := stOutlet_Valve_Int.bCmdWP,
    i_ServiceMode := stOutlet_Valve_Int.bServiceMode,
    i_EnableHP := stOutlet_Valve_Int.bEnableHP,
    i_EnableWP := stOutlet_Valve_Int.bEnableWP,
    i_HP := IN.bOutletPos_Opened,
    i_WP := IN.bOutletPos_Closed,
    i_Timeout := stOutlet_Valve_Int.iTravelTimeout,
    i_MaintLimit := stOutlet_Valve_Int.iMaintLimit,
    i_PresetValue := stOutlet_Valve_Int.iPresetValue,
    i_WritePreset := stOutlet_Valve_Int.bWritePreset,
    q_InterlocksOK => stOutlet_Valve_Int.bInterlocksOK,
    q_CmdWP => stOutlet_Valve_Int.bCmdOutWP,
    q_TotalCycles => stOutlet_Valve_Int.iTotalCycles,
    q_MaintCycles => stOutlet_Valve_Int.iMaintCycles,
    q_MaintenanceCall => stOutlet_Valve_Int.bMaintCall,
    q_State => stOutlet_Valve_Int.iState); // FB_ValveCtrl52
stOutlet_Valve_Int.bCmdOutHP := fbOutlet_Valve.q_CmdHP;

// NETWORK 4
OUT.bOutlet_Valve_Open := stOutlet_Valve_Int.bCmdOutHP;

// NETWORK 5
OUT.bOutlet_Valve_Close := stOutlet_Valve_Int.bCmdOutWP;

// NETWORK 6
stOutlet_Valve_Int.arrInterlocks := F_ToArrInterlocks(In1 := TRUE, In2 := TRUE, In3 := TRUE, In4 := TRUE, In5 := TRUE, In6 := TRUE, In7 := TRUE, In8 := TRUE);

// NETWORK 7
stOutlet_Valve_Int.arrAlarms := F_ToArrAlarms(In1 := fbOutlet_Valve.q_TimeoutHP, In2 := fbOutlet_Valve.q_TimeoutWP, In3 := fbOutlet_Valve.q_SensorsFlt, In4 := FALSE, In5 := FALSE, In6 := FALSE, In7 := FALSE, In8 := FALSE, AlarmsNOK => stOutlet_Valve_Int.bFault);

// NETWORK 8
_w4 := NOT stOutlet_Valve_Int.bServiceMode;
stOutlet_Valve_Int.bCmdHP R= _w4;
stOutlet_Valve_Int.bCmdWP R= _w4;

// NETWORK 9
OUT.bOutletOpen_Light := IN.bOutletPos_Opened;

// NETWORK 10
OUT.bOutletClose_Light := IN.bOutletPos_Closed;
END_ACTION

ACTION PROD_AirSeal:
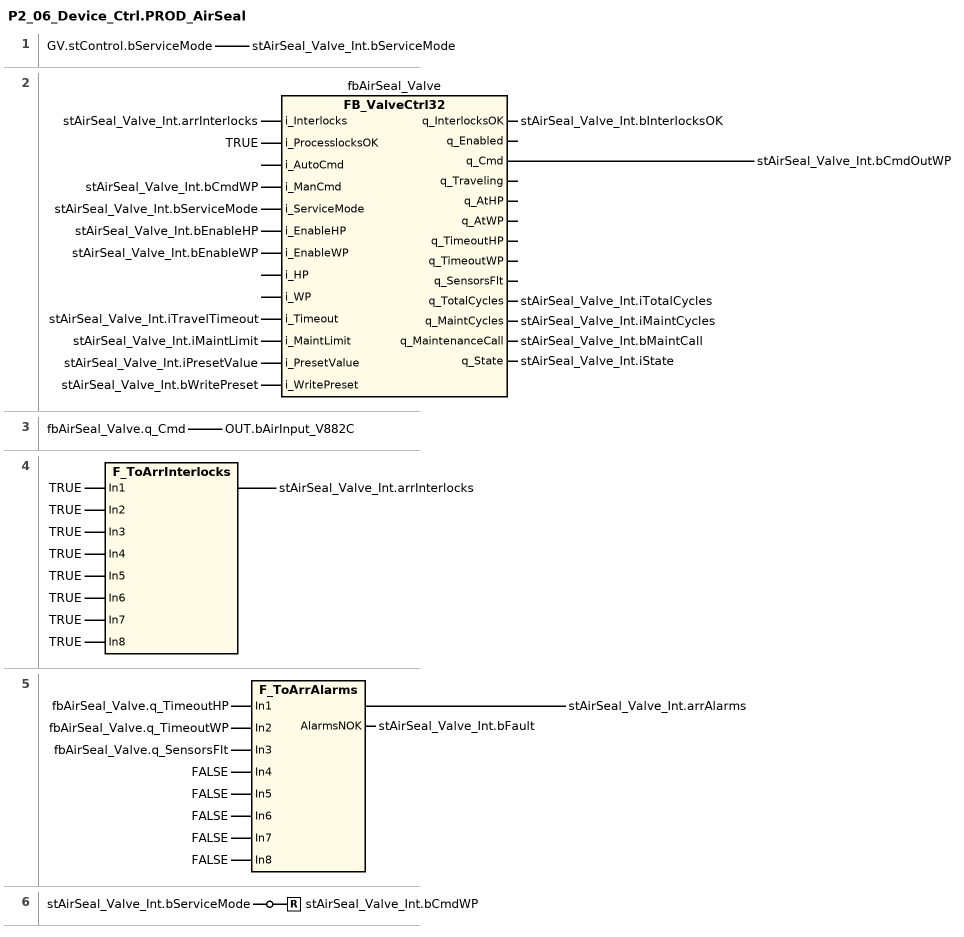
// NETWORK 1
stAirSeal_Valve_Int.bServiceMode := GV.stControl.bServiceMode;

// NETWORK 2
fbAirSeal_Valve(
    i_Interlocks := stAirSeal_Valve_Int.arrInterlocks,
    i_ProcesslocksOK := TRUE,
    i_ManCmd := stAirSeal_Valve_Int.bCmdWP,
    i_ServiceMode := stAirSeal_Valve_Int.bServiceMode,
    i_EnableHP := stAirSeal_Valve_Int.bEnableHP,
    i_EnableWP := stAirSeal_Valve_Int.bEnableWP,
    i_Timeout := stAirSeal_Valve_Int.iTravelTimeout,
    i_MaintLimit := stAirSeal_Valve_Int.iMaintLimit,
    i_PresetValue := stAirSeal_Valve_Int.iPresetValue,
    i_WritePreset := stAirSeal_Valve_Int.bWritePreset,
    q_InterlocksOK => stAirSeal_Valve_Int.bInterlocksOK,
    q_TotalCycles => stAirSeal_Valve_Int.iTotalCycles,
    q_MaintCycles => stAirSeal_Valve_Int.iMaintCycles,
    q_MaintenanceCall => stAirSeal_Valve_Int.bMaintCall,
    q_State => stAirSeal_Valve_Int.iState); // FB_ValveCtrl32
stAirSeal_Valve_Int.bCmdOutWP := fbAirSeal_Valve.q_Cmd;

// NETWORK 3
OUT.bAirInput_V882C := fbAirSeal_Valve.q_Cmd;

// NETWORK 4
stAirSeal_Valve_Int.arrInterlocks := F_ToArrInterlocks(In1 := TRUE, In2 := TRUE, In3 := TRUE, In4 := TRUE, In5 := TRUE, In6 := TRUE, In7 := TRUE, In8 := TRUE);

// NETWORK 5
stAirSeal_Valve_Int.arrAlarms := F_ToArrAlarms(In1 := fbAirSeal_Valve.q_TimeoutHP, In2 := fbAirSeal_Valve.q_TimeoutWP, In3 := fbAirSeal_Valve.q_SensorsFlt, In4 := FALSE, In5 := FALSE, In6 := FALSE, In7 := FALSE, In8 := FALSE, AlarmsNOK => stAirSeal_Valve_Int.bFault);

// NETWORK 6
stAirSeal_Valve_Int.bCmdWP R= NOT stAirSeal_Valve_Int.bServiceMode;
END_ACTION

ACTION PROD_Aspiration:
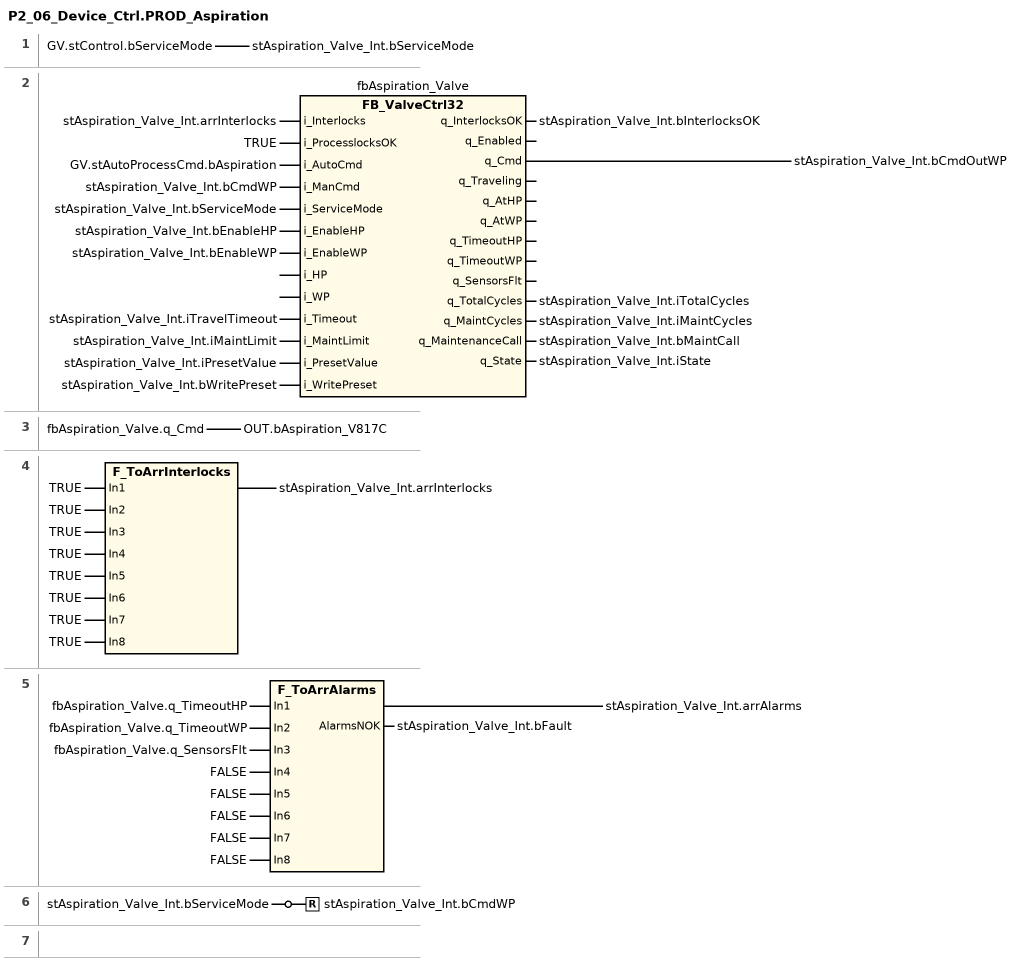
// NETWORK 1
stAspiration_Valve_Int.bServiceMode := GV.stControl.bServiceMode;

// NETWORK 2
fbAspiration_Valve(
    i_Interlocks := stAspiration_Valve_Int.arrInterlocks,
    i_ProcesslocksOK := TRUE,
    i_AutoCmd := GV.stAutoProcessCmd.bAspiration,
    i_ManCmd := stAspiration_Valve_Int.bCmdWP,
    i_ServiceMode := stAspiration_Valve_Int.bServiceMode,
    i_EnableHP := stAspiration_Valve_Int.bEnableHP,
    i_EnableWP := stAspiration_Valve_Int.bEnableWP,
    i_Timeout := stAspiration_Valve_Int.iTravelTimeout,
    i_MaintLimit := stAspiration_Valve_Int.iMaintLimit,
    i_PresetValue := stAspiration_Valve_Int.iPresetValue,
    i_WritePreset := stAspiration_Valve_Int.bWritePreset,
    q_InterlocksOK => stAspiration_Valve_Int.bInterlocksOK,
    q_TotalCycles => stAspiration_Valve_Int.iTotalCycles,
    q_MaintCycles => stAspiration_Valve_Int.iMaintCycles,
    q_MaintenanceCall => stAspiration_Valve_Int.bMaintCall,
    q_State => stAspiration_Valve_Int.iState); // FB_ValveCtrl32
stAspiration_Valve_Int.bCmdOutWP := fbAspiration_Valve.q_Cmd;

// NETWORK 3
OUT.bAspiration_V817C := fbAspiration_Valve.q_Cmd;

// NETWORK 4
stAspiration_Valve_Int.arrInterlocks := F_ToArrInterlocks(In1 := TRUE, In2 := TRUE, In3 := TRUE, In4 := TRUE, In5 := TRUE, In6 := TRUE, In7 := TRUE, In8 := TRUE);

// NETWORK 5
stAspiration_Valve_Int.arrAlarms := F_ToArrAlarms(In1 := fbAspiration_Valve.q_TimeoutHP, In2 := fbAspiration_Valve.q_TimeoutWP, In3 := fbAspiration_Valve.q_SensorsFlt, In4 := FALSE, In5 := FALSE, In6 := FALSE, In7 := FALSE, In8 := FALSE, AlarmsNOK => stAspiration_Valve_Int.bFault);

// NETWORK 6
stAspiration_Valve_Int.bCmdWP R= NOT stAspiration_Valve_Int.bServiceMode;

// NETWORK 7
END_ACTION

ACTION PROD_ChopperAir:
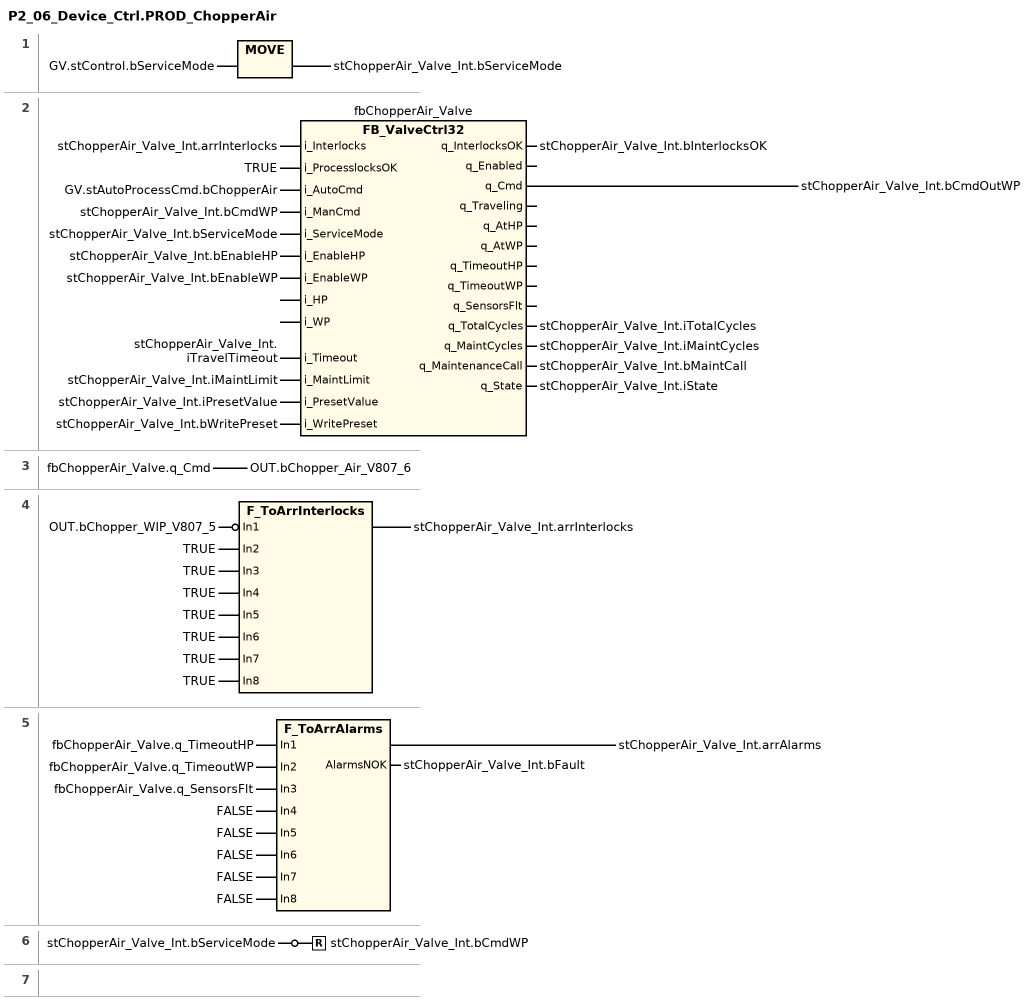
// NETWORK 1
stChopperAir_Valve_Int.bServiceMode := GV.stControl.bServiceMode;

// NETWORK 2
fbChopperAir_Valve(
    i_Interlocks := stChopperAir_Valve_Int.arrInterlocks,
    i_ProcesslocksOK := TRUE,
    i_AutoCmd := GV.stAutoProcessCmd.bChopperAir,
    i_ManCmd := stChopperAir_Valve_Int.bCmdWP,
    i_ServiceMode := stChopperAir_Valve_Int.bServiceMode,
    i_EnableHP := stChopperAir_Valve_Int.bEnableHP,
    i_EnableWP := stChopperAir_Valve_Int.bEnableWP,
    i_Timeout := stChopperAir_Valve_Int.iTravelTimeout,
    i_MaintLimit := stChopperAir_Valve_Int.iMaintLimit,
    i_PresetValue := stChopperAir_Valve_Int.iPresetValue,
    i_WritePreset := stChopperAir_Valve_Int.bWritePreset,
    q_InterlocksOK => stChopperAir_Valve_Int.bInterlocksOK,
    q_TotalCycles => stChopperAir_Valve_Int.iTotalCycles,
    q_MaintCycles => stChopperAir_Valve_Int.iMaintCycles,
    q_MaintenanceCall => stChopperAir_Valve_Int.bMaintCall,
    q_State => stChopperAir_Valve_Int.iState); // FB_ValveCtrl32
stChopperAir_Valve_Int.bCmdOutWP := fbChopperAir_Valve.q_Cmd;

// NETWORK 3
OUT.bChopper_Air_V807_6 := fbChopperAir_Valve.q_Cmd;

// NETWORK 4
stChopperAir_Valve_Int.arrInterlocks := F_ToArrInterlocks(In1 := NOT OUT.bChopper_WIP_V807_5, In2 := TRUE, In3 := TRUE, In4 := TRUE, In5 := TRUE, In6 := TRUE, In7 := TRUE, In8 := TRUE);

// NETWORK 5
stChopperAir_Valve_Int.arrAlarms := F_ToArrAlarms(In1 := fbChopperAir_Valve.q_TimeoutHP, In2 := fbChopperAir_Valve.q_TimeoutWP, In3 := fbChopperAir_Valve.q_SensorsFlt, In4 := FALSE, In5 := FALSE, In6 := FALSE, In7 := FALSE, In8 := FALSE, AlarmsNOK => stChopperAir_Valve_Int.bFault);

// NETWORK 6
stChopperAir_Valve_Int.bCmdWP R= NOT stChopperAir_Valve_Int.bServiceMode;

// NETWORK 7
END_ACTION

ACTION PROD_FilterClean:
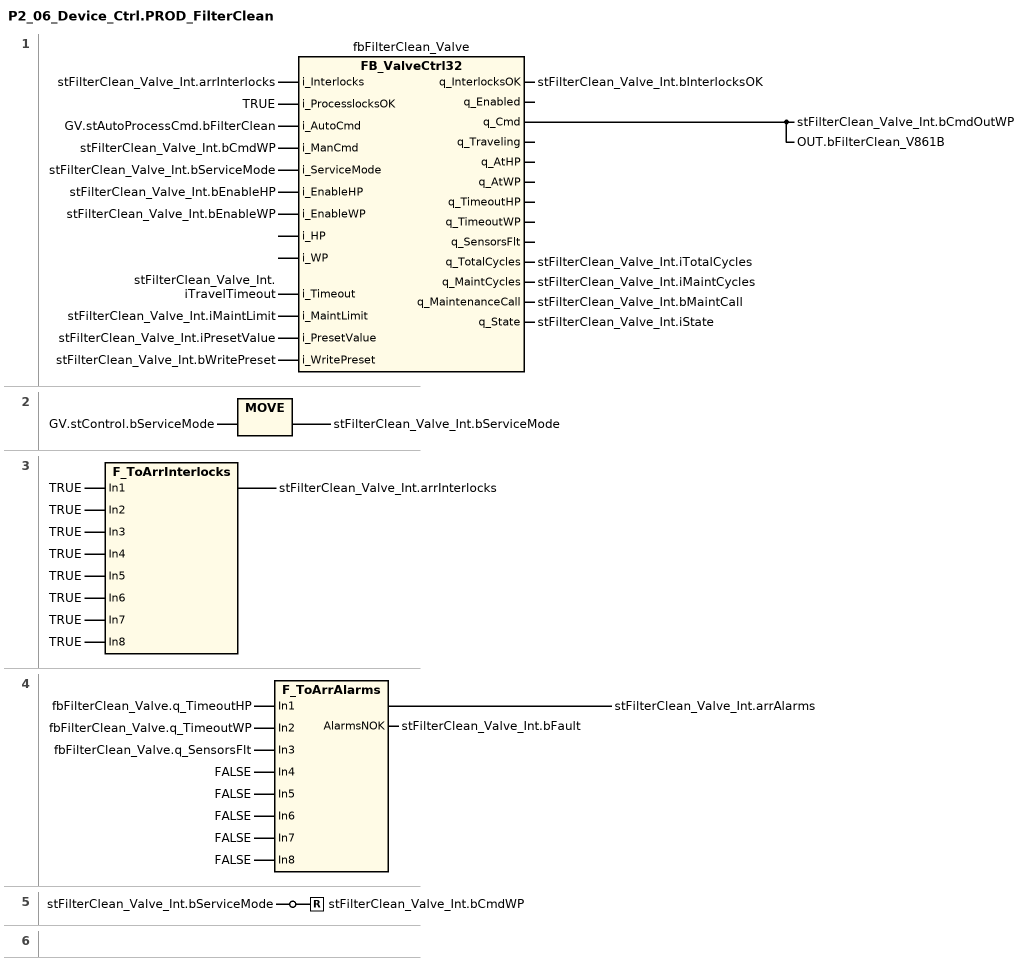
// NETWORK 1
fbFilterClean_Valve(
    i_Interlocks := stFilterClean_Valve_Int.arrInterlocks,
    i_ProcesslocksOK := TRUE,
    i_AutoCmd := GV.stAutoProcessCmd.bFilterClean,
    i_ManCmd := stFilterClean_Valve_Int.bCmdWP,
    i_ServiceMode := stFilterClean_Valve_Int.bServiceMode,
    i_EnableHP := stFilterClean_Valve_Int.bEnableHP,
    i_EnableWP := stFilterClean_Valve_Int.bEnableWP,
    i_Timeout := stFilterClean_Valve_Int.iTravelTimeout,
    i_MaintLimit := stFilterClean_Valve_Int.iMaintLimit,
    i_PresetValue := stFilterClean_Valve_Int.iPresetValue,
    i_WritePreset := stFilterClean_Valve_Int.bWritePreset,
    q_InterlocksOK => stFilterClean_Valve_Int.bInterlocksOK,
    q_TotalCycles => stFilterClean_Valve_Int.iTotalCycles,
    q_MaintCycles => stFilterClean_Valve_Int.iMaintCycles,
    q_MaintenanceCall => stFilterClean_Valve_Int.bMaintCall,
    q_State => stFilterClean_Valve_Int.iState); // FB_ValveCtrl32
stFilterClean_Valve_Int.bCmdOutWP := fbFilterClean_Valve.q_Cmd;
OUT.bFilterClean_V861B := fbFilterClean_Valve.q_Cmd;

// NETWORK 2
stFilterClean_Valve_Int.bServiceMode := GV.stControl.bServiceMode;

// NETWORK 3
stFilterClean_Valve_Int.arrInterlocks := F_ToArrInterlocks(In1 := TRUE, In2 := TRUE, In3 := TRUE, In4 := TRUE, In5 := TRUE, In6 := TRUE, In7 := TRUE, In8 := TRUE);

// NETWORK 4
stFilterClean_Valve_Int.arrAlarms := F_ToArrAlarms(In1 := fbFilterClean_Valve.q_TimeoutHP, In2 := fbFilterClean_Valve.q_TimeoutWP, In3 := fbFilterClean_Valve.q_SensorsFlt, In4 := FALSE, In5 := FALSE, In6 := FALSE, In7 := FALSE, In8 := FALSE, AlarmsNOK => stFilterClean_Valve_Int.bFault);

// NETWORK 5
stFilterClean_Valve_Int.bCmdWP R= NOT stFilterClean_Valve_Int.bServiceMode;

// NETWORK 6
END_ACTION

ACTION PROD_MixerAir:
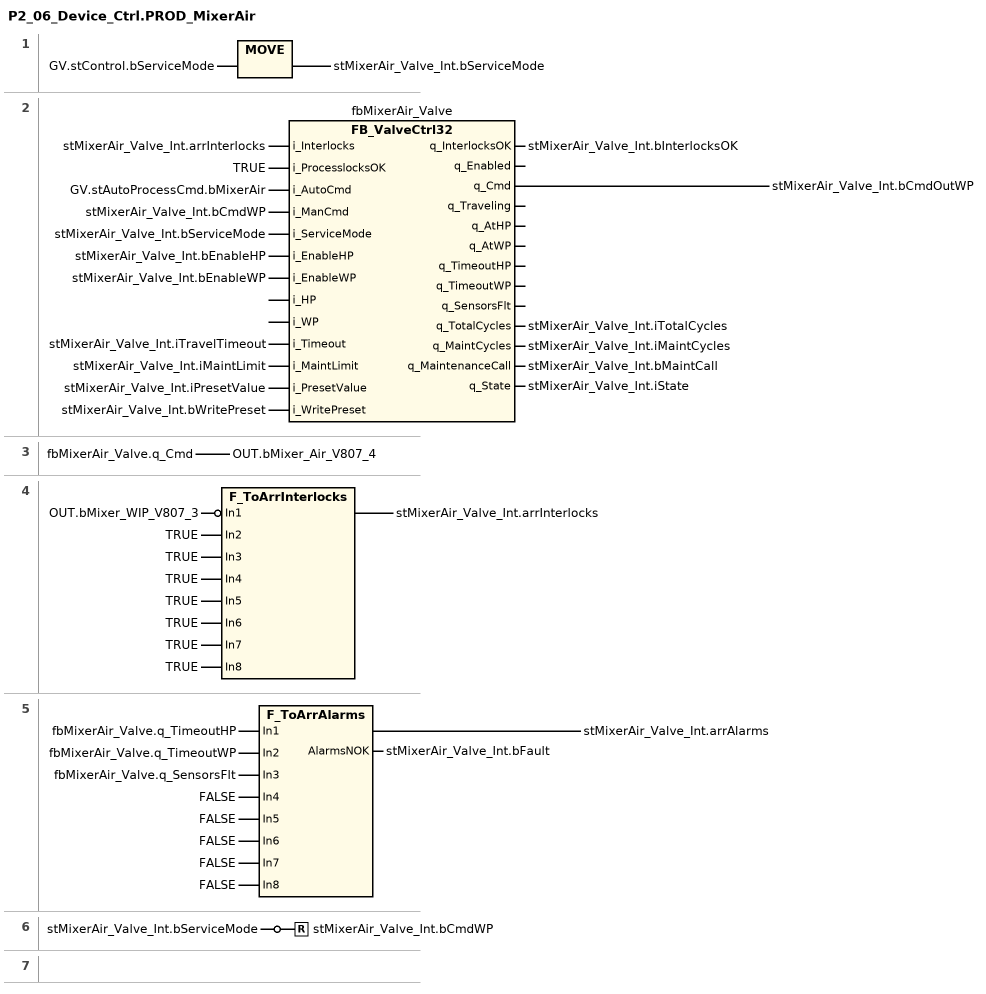
// NETWORK 1
stMixerAir_Valve_Int.bServiceMode := GV.stControl.bServiceMode;

// NETWORK 2
fbMixerAir_Valve(
    i_Interlocks := stMixerAir_Valve_Int.arrInterlocks,
    i_ProcesslocksOK := TRUE,
    i_AutoCmd := GV.stAutoProcessCmd.bMixerAir,
    i_ManCmd := stMixerAir_Valve_Int.bCmdWP,
    i_ServiceMode := stMixerAir_Valve_Int.bServiceMode,
    i_EnableHP := stMixerAir_Valve_Int.bEnableHP,
    i_EnableWP := stMixerAir_Valve_Int.bEnableWP,
    i_Timeout := stMixerAir_Valve_Int.iTravelTimeout,
    i_MaintLimit := stMixerAir_Valve_Int.iMaintLimit,
    i_PresetValue := stMixerAir_Valve_Int.iPresetValue,
    i_WritePreset := stMixerAir_Valve_Int.bWritePreset,
    q_InterlocksOK => stMixerAir_Valve_Int.bInterlocksOK,
    q_TotalCycles => stMixerAir_Valve_Int.iTotalCycles,
    q_MaintCycles => stMixerAir_Valve_Int.iMaintCycles,
    q_MaintenanceCall => stMixerAir_Valve_Int.bMaintCall,
    q_State => stMixerAir_Valve_Int.iState); // FB_ValveCtrl32
stMixerAir_Valve_Int.bCmdOutWP := fbMixerAir_Valve.q_Cmd;

// NETWORK 3
OUT.bMixer_Air_V807_4 := fbMixerAir_Valve.q_Cmd;

// NETWORK 4
stMixerAir_Valve_Int.arrInterlocks := F_ToArrInterlocks(In1 := NOT OUT.bMixer_WIP_V807_3, In2 := TRUE, In3 := TRUE, In4 := TRUE, In5 := TRUE, In6 := TRUE, In7 := TRUE, In8 := TRUE);

// NETWORK 5
stMixerAir_Valve_Int.arrAlarms := F_ToArrAlarms(In1 := fbMixerAir_Valve.q_TimeoutHP, In2 := fbMixerAir_Valve.q_TimeoutWP, In3 := fbMixerAir_Valve.q_SensorsFlt, In4 := FALSE, In5 := FALSE, In6 := FALSE, In7 := FALSE, In8 := FALSE, AlarmsNOK => stMixerAir_Valve_Int.bFault);

// NETWORK 6
stMixerAir_Valve_Int.bCmdWP R= NOT stMixerAir_Valve_Int.bServiceMode;

// NETWORK 7
END_ACTION

ACTION PROD_Vacuum:
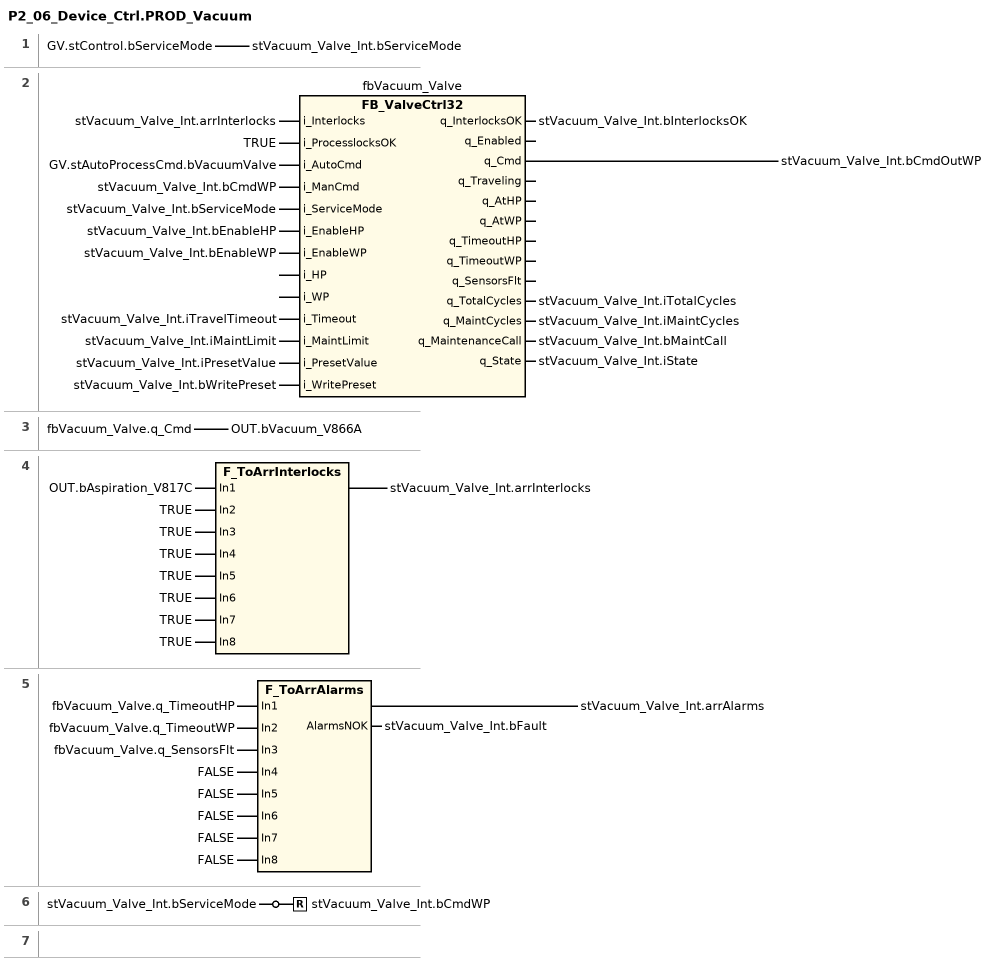
// NETWORK 1
stVacuum_Valve_Int.bServiceMode := GV.stControl.bServiceMode;

// NETWORK 2
fbVacuum_Valve(
    i_Interlocks := stVacuum_Valve_Int.arrInterlocks,
    i_ProcesslocksOK := TRUE,
    i_AutoCmd := GV.stAutoProcessCmd.bVacuumValve,
    i_ManCmd := stVacuum_Valve_Int.bCmdWP,
    i_ServiceMode := stVacuum_Valve_Int.bServiceMode,
    i_EnableHP := stVacuum_Valve_Int.bEnableHP,
    i_EnableWP := stVacuum_Valve_Int.bEnableWP,
    i_Timeout := stVacuum_Valve_Int.iTravelTimeout,
    i_MaintLimit := stVacuum_Valve_Int.iMaintLimit,
    i_PresetValue := stVacuum_Valve_Int.iPresetValue,
    i_WritePreset := stVacuum_Valve_Int.bWritePreset,
    q_InterlocksOK => stVacuum_Valve_Int.bInterlocksOK,
    q_TotalCycles => stVacuum_Valve_Int.iTotalCycles,
    q_MaintCycles => stVacuum_Valve_Int.iMaintCycles,
    q_MaintenanceCall => stVacuum_Valve_Int.bMaintCall,
    q_State => stVacuum_Valve_Int.iState); // FB_ValveCtrl32
stVacuum_Valve_Int.bCmdOutWP := fbVacuum_Valve.q_Cmd;

// NETWORK 3
OUT.bVacuum_V866A := fbVacuum_Valve.q_Cmd;

// NETWORK 4
stVacuum_Valve_Int.arrInterlocks := F_ToArrInterlocks(In1 := OUT.bAspiration_V817C, In2 := TRUE, In3 := TRUE, In4 := TRUE, In5 := TRUE, In6 := TRUE, In7 := TRUE, In8 := TRUE);

// NETWORK 5
stVacuum_Valve_Int.arrAlarms := F_ToArrAlarms(In1 := fbVacuum_Valve.q_TimeoutHP, In2 := fbVacuum_Valve.q_TimeoutWP, In3 := fbVacuum_Valve.q_SensorsFlt, In4 := FALSE, In5 := FALSE, In6 := FALSE, In7 := FALSE, In8 := FALSE, AlarmsNOK => stVacuum_Valve_Int.bFault);

// NETWORK 6
stVacuum_Valve_Int.bCmdWP R= NOT stVacuum_Valve_Int.bServiceMode;

// NETWORK 7
END_ACTION

ACTION Pump:
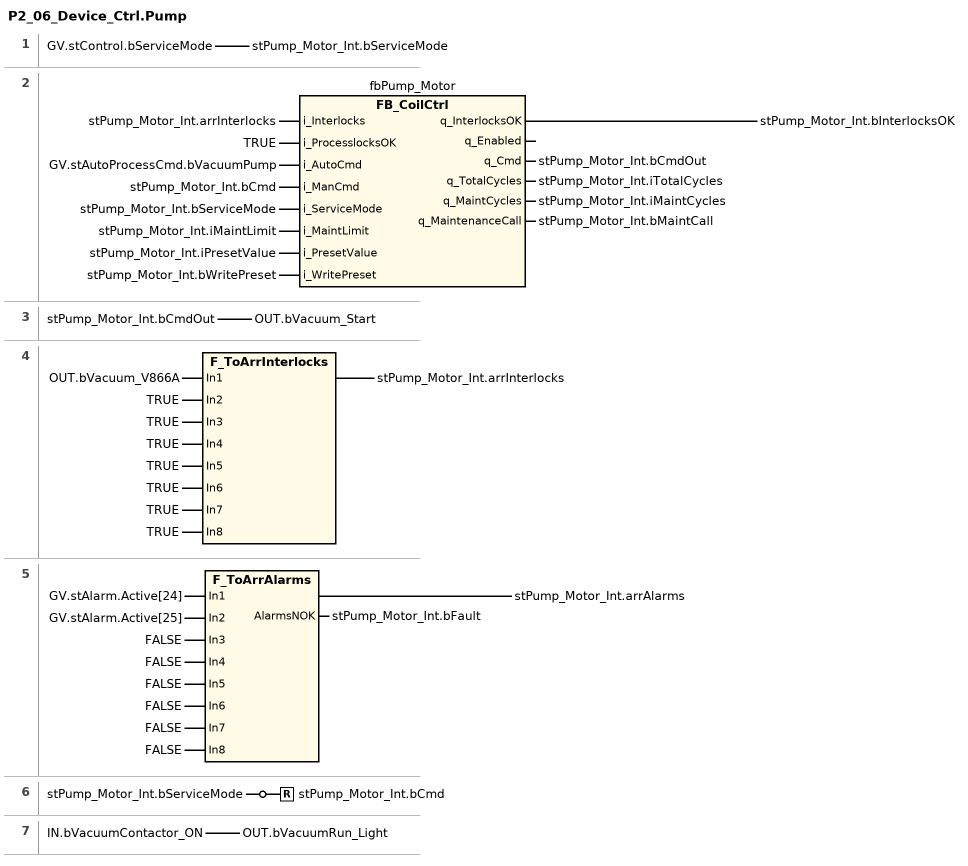
// NETWORK 1
stPump_Motor_Int.bServiceMode := GV.stControl.bServiceMode;

// NETWORK 2
fbPump_Motor(
    i_Interlocks := stPump_Motor_Int.arrInterlocks,
    i_ProcesslocksOK := TRUE,
    i_AutoCmd := GV.stAutoProcessCmd.bVacuumPump,
    i_ManCmd := stPump_Motor_Int.bCmd,
    i_ServiceMode := stPump_Motor_Int.bServiceMode,
    i_MaintLimit := stPump_Motor_Int.iMaintLimit,
    i_PresetValue := stPump_Motor_Int.iPresetValue,
    i_WritePreset := stPump_Motor_Int.bWritePreset,
    q_Cmd => stPump_Motor_Int.bCmdOut,
    q_TotalCycles => stPump_Motor_Int.iTotalCycles,
    q_MaintCycles => stPump_Motor_Int.iMaintCycles,
    q_MaintenanceCall => stPump_Motor_Int.bMaintCall); // FB_CoilCtrl
stPump_Motor_Int.bInterlocksOK := fbPump_Motor.q_InterlocksOK;

// NETWORK 3
OUT.bVacuum_Start := stPump_Motor_Int.bCmdOut;

// NETWORK 4
stPump_Motor_Int.arrInterlocks := F_ToArrInterlocks(In1 := OUT.bVacuum_V866A, In2 := TRUE, In3 := TRUE, In4 := TRUE, In5 := TRUE, In6 := TRUE, In7 := TRUE, In8 := TRUE);

// NETWORK 5
stPump_Motor_Int.arrAlarms := F_ToArrAlarms(In1 := GV.stAlarm.Active[24], In2 := GV.stAlarm.Active[25], In3 := FALSE, In4 := FALSE, In5 := FALSE, In6 := FALSE, In7 := FALSE, In8 := FALSE, AlarmsNOK => stPump_Motor_Int.bFault);

// NETWORK 6
stPump_Motor_Int.bCmd R= NOT stPump_Motor_Int.bServiceMode;

// NETWORK 7
OUT.bVacuumRun_Light := IN.bVacuumContactor_ON;
END_ACTION

ACTION Purge:
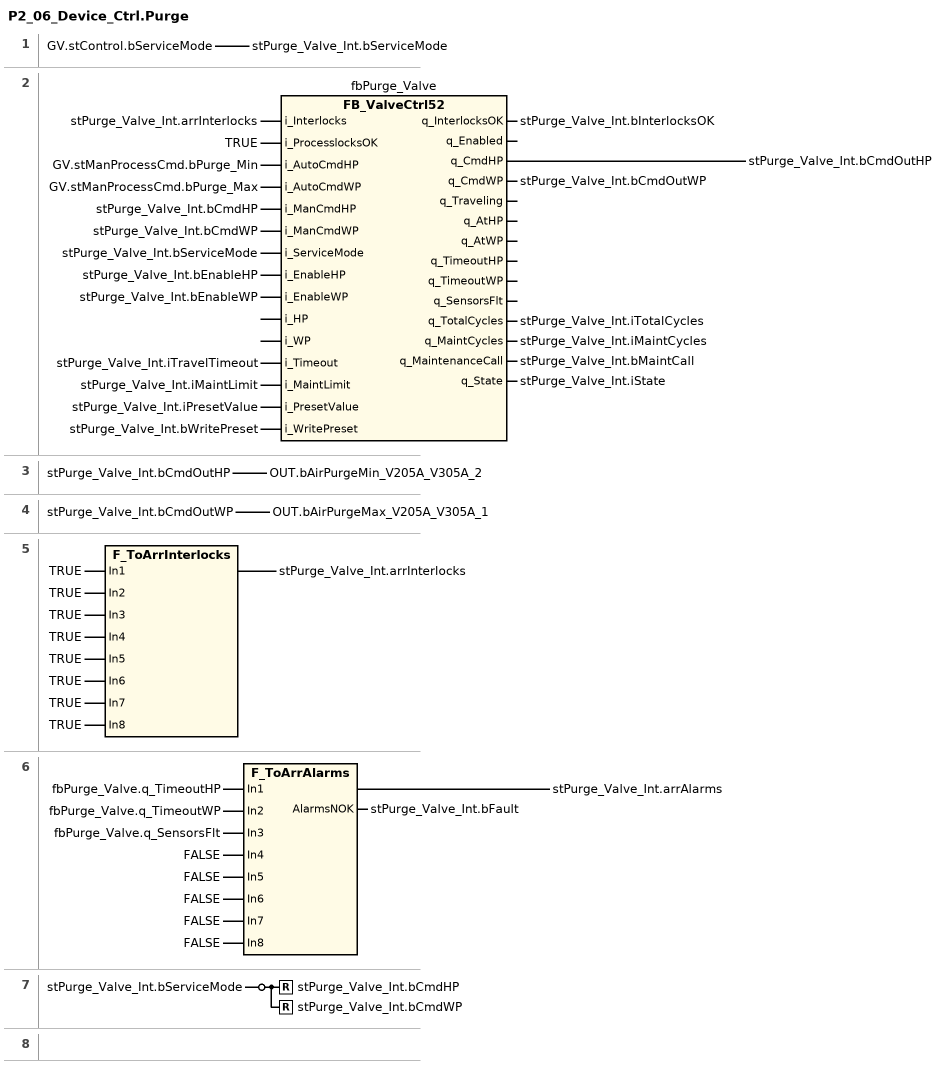
// NETWORK 1
stPurge_Valve_Int.bServiceMode := GV.stControl.bServiceMode;

// NETWORK 2
fbPurge_Valve(
    i_Interlocks := stPurge_Valve_Int.arrInterlocks,
    i_ProcesslocksOK := TRUE,
    i_AutoCmdHP := GV.stManProcessCmd.bPurge_Min,
    i_AutoCmdWP := GV.stManProcessCmd.bPurge_Max,
    i_ManCmdHP := stPurge_Valve_Int.bCmdHP,
    i_ManCmdWP := stPurge_Valve_Int.bCmdWP,
    i_ServiceMode := stPurge_Valve_Int.bServiceMode,
    i_EnableHP := stPurge_Valve_Int.bEnableHP,
    i_EnableWP := stPurge_Valve_Int.bEnableWP,
    i_Timeout := stPurge_Valve_Int.iTravelTimeout,
    i_MaintLimit := stPurge_Valve_Int.iMaintLimit,
    i_PresetValue := stPurge_Valve_Int.iPresetValue,
    i_WritePreset := stPurge_Valve_Int.bWritePreset,
    q_InterlocksOK => stPurge_Valve_Int.bInterlocksOK,
    q_CmdWP => stPurge_Valve_Int.bCmdOutWP,
    q_TotalCycles => stPurge_Valve_Int.iTotalCycles,
    q_MaintCycles => stPurge_Valve_Int.iMaintCycles,
    q_MaintenanceCall => stPurge_Valve_Int.bMaintCall,
    q_State => stPurge_Valve_Int.iState); // FB_ValveCtrl52
stPurge_Valve_Int.bCmdOutHP := fbPurge_Valve.q_CmdHP;

// NETWORK 3
OUT.bAirPurgeMin_V205A_V305A_2 := stPurge_Valve_Int.bCmdOutHP;

// NETWORK 4
OUT.bAirPurgeMax_V205A_V305A_1 := stPurge_Valve_Int.bCmdOutWP;

// NETWORK 5
stPurge_Valve_Int.arrInterlocks := F_ToArrInterlocks(In1 := TRUE, In2 := TRUE, In3 := TRUE, In4 := TRUE, In5 := TRUE, In6 := TRUE, In7 := TRUE, In8 := TRUE);

// NETWORK 6
stPurge_Valve_Int.arrAlarms := F_ToArrAlarms(In1 := fbPurge_Valve.q_TimeoutHP, In2 := fbPurge_Valve.q_TimeoutWP, In3 := fbPurge_Valve.q_SensorsFlt, In4 := FALSE, In5 := FALSE, In6 := FALSE, In7 := FALSE, In8 := FALSE, AlarmsNOK => stPurge_Valve_Int.bFault);

// NETWORK 7
_w5 := NOT stPurge_Valve_Int.bServiceMode;
stPurge_Valve_Int.bCmdHP R= _w5;
stPurge_Valve_Int.bCmdWP R= _w5;

// NETWORK 8
END_ACTION

ACTION Seal:
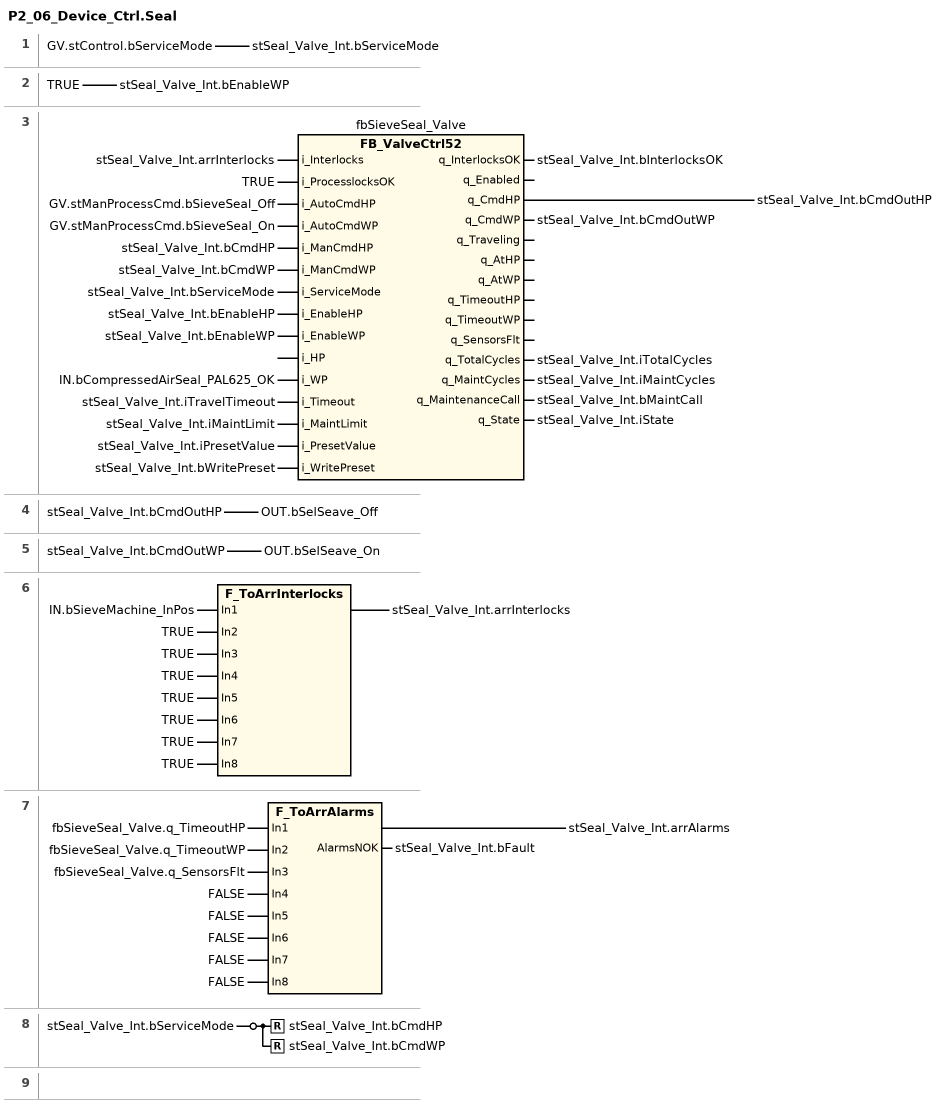
// NETWORK 1
stSeal_Valve_Int.bServiceMode := GV.stControl.bServiceMode;

// NETWORK 2
stSeal_Valve_Int.bEnableWP := TRUE;

// NETWORK 3
fbSieveSeal_Valve(
    i_Interlocks := stSeal_Valve_Int.arrInterlocks,
    i_ProcesslocksOK := TRUE,
    i_AutoCmdHP := GV.stManProcessCmd.bSieveSeal_Off,
    i_AutoCmdWP := GV.stManProcessCmd.bSieveSeal_On,
    i_ManCmdHP := stSeal_Valve_Int.bCmdHP,
    i_ManCmdWP := stSeal_Valve_Int.bCmdWP,
    i_ServiceMode := stSeal_Valve_Int.bServiceMode,
    i_EnableHP := stSeal_Valve_Int.bEnableHP,
    i_EnableWP := stSeal_Valve_Int.bEnableWP,
    i_WP := IN.bCompressedAirSeal_PAL625_OK,
    i_Timeout := stSeal_Valve_Int.iTravelTimeout,
    i_MaintLimit := stSeal_Valve_Int.iMaintLimit,
    i_PresetValue := stSeal_Valve_Int.iPresetValue,
    i_WritePreset := stSeal_Valve_Int.bWritePreset,
    q_InterlocksOK => stSeal_Valve_Int.bInterlocksOK,
    q_CmdWP => stSeal_Valve_Int.bCmdOutWP,
    q_TotalCycles => stSeal_Valve_Int.iTotalCycles,
    q_MaintCycles => stSeal_Valve_Int.iMaintCycles,
    q_MaintenanceCall => stSeal_Valve_Int.bMaintCall,
    q_State => stSeal_Valve_Int.iState); // FB_ValveCtrl52
stSeal_Valve_Int.bCmdOutHP := fbSieveSeal_Valve.q_CmdHP;

// NETWORK 4
OUT.bSelSeave_Off := stSeal_Valve_Int.bCmdOutHP;

// NETWORK 5
OUT.bSelSeave_On := stSeal_Valve_Int.bCmdOutWP;

// NETWORK 6
stSeal_Valve_Int.arrInterlocks := F_ToArrInterlocks(In1 := IN.bSieveMachine_InPos, In2 := TRUE, In3 := TRUE, In4 := TRUE, In5 := TRUE, In6 := TRUE, In7 := TRUE, In8 := TRUE);

// NETWORK 7
stSeal_Valve_Int.arrAlarms := F_ToArrAlarms(In1 := fbSieveSeal_Valve.q_TimeoutHP, In2 := fbSieveSeal_Valve.q_TimeoutWP, In3 := fbSieveSeal_Valve.q_SensorsFlt, In4 := FALSE, In5 := FALSE, In6 := FALSE, In7 := FALSE, In8 := FALSE, AlarmsNOK => stSeal_Valve_Int.bFault);

// NETWORK 8
_w6 := NOT stSeal_Valve_Int.bServiceMode;
stSeal_Valve_Int.bCmdHP R= _w6;
stSeal_Valve_Int.bCmdWP R= _w6;

// NETWORK 9
END_ACTION

ACTION Sieve:
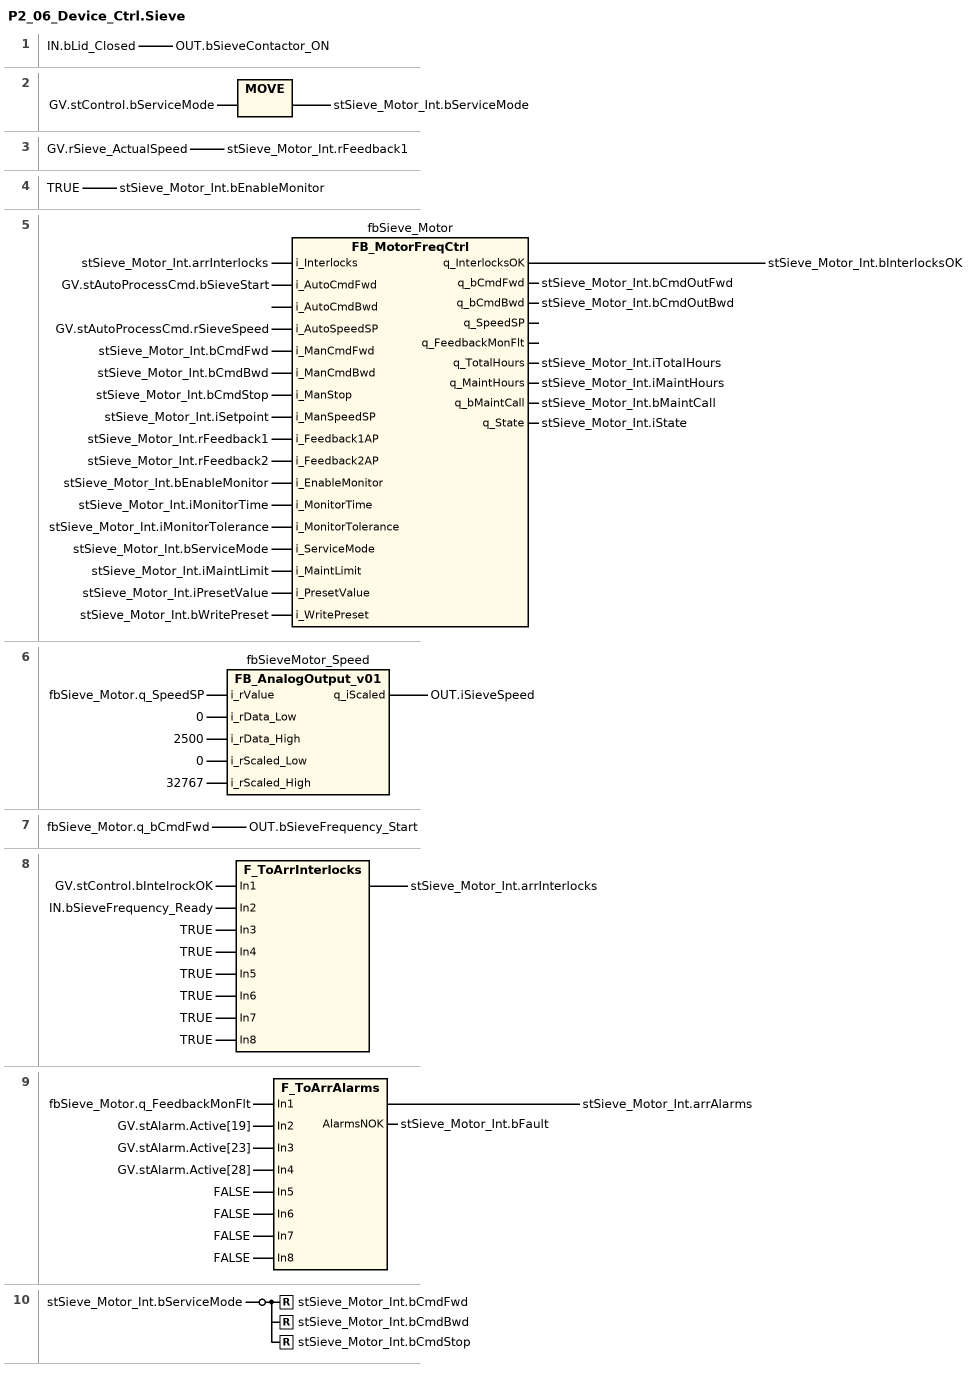
// NETWORK 1
OUT.bSieveContactor_ON := IN.bLid_Closed;

// NETWORK 2
stSieve_Motor_Int.bServiceMode := GV.stControl.bServiceMode;

// NETWORK 3
stSieve_Motor_Int.rFeedback1 := GV.rSieve_ActualSpeed;

// NETWORK 4
stSieve_Motor_Int.bEnableMonitor := TRUE;

// NETWORK 5
fbSieve_Motor(
    i_Interlocks := stSieve_Motor_Int.arrInterlocks,
    i_AutoCmdFwd := GV.stAutoProcessCmd.bSieveStart,
    i_AutoSpeedSP := GV.stAutoProcessCmd.rSieveSpeed,
    i_ManCmdFwd := stSieve_Motor_Int.bCmdFwd,
    i_ManCmdBwd := stSieve_Motor_Int.bCmdBwd,
    i_ManStop := stSieve_Motor_Int.bCmdStop,
    i_ManSpeedSP := stSieve_Motor_Int.iSetpoint,
    i_Feedback1AP := stSieve_Motor_Int.rFeedback1,
    i_Feedback2AP := stSieve_Motor_Int.rFeedback2,
    i_EnableMonitor := stSieve_Motor_Int.bEnableMonitor,
    i_MonitorTime := stSieve_Motor_Int.iMonitorTime,
    i_MonitorTolerance := stSieve_Motor_Int.iMonitorTolerance,
    i_ServiceMode := stSieve_Motor_Int.bServiceMode,
    i_MaintLimit := stSieve_Motor_Int.iMaintLimit,
    i_PresetValue := stSieve_Motor_Int.iPresetValue,
    i_WritePreset := stSieve_Motor_Int.bWritePreset,
    q_bCmdFwd => stSieve_Motor_Int.bCmdOutFwd,
    q_bCmdBwd => stSieve_Motor_Int.bCmdOutBwd,
    q_TotalHours => stSieve_Motor_Int.iTotalHours,
    q_MaintHours => stSieve_Motor_Int.iMaintHours,
    q_bMaintCall => stSieve_Motor_Int.bMaintCall,
    q_State => stSieve_Motor_Int.iState); // FB_MotorFreqCtrl
stSieve_Motor_Int.bInterlocksOK := fbSieve_Motor.q_InterlocksOK;

// NETWORK 6
fbSieveMotor_Speed(
    i_rValue := fbSieve_Motor.q_SpeedSP,
    i_rData_Low := 0,
    i_rData_High := 2500,
    i_rScaled_Low := 0,
    i_rScaled_High := 32767); // FB_AnalogOutput_v01
OUT.iSieveSpeed := fbSieveMotor_Speed.q_iScaled;

// NETWORK 7
OUT.bSieveFrequency_Start := fbSieve_Motor.q_bCmdFwd;

// NETWORK 8
stSieve_Motor_Int.arrInterlocks := F_ToArrInterlocks(In1 := GV.stControl.bIntelrockOK, In2 := IN.bSieveFrequency_Ready, In3 := TRUE, In4 := TRUE, In5 := TRUE, In6 := TRUE, In7 := TRUE, In8 := TRUE);

// NETWORK 9
stSieve_Motor_Int.arrAlarms := F_ToArrAlarms(In1 := fbSieve_Motor.q_FeedbackMonFlt, In2 := GV.stAlarm.Active[19], In3 := GV.stAlarm.Active[23], In4 := GV.stAlarm.Active[28], In5 := FALSE, In6 := FALSE, In7 := FALSE, In8 := FALSE, AlarmsNOK => stSieve_Motor_Int.bFault);

// NETWORK 10
_w7 := NOT stSieve_Motor_Int.bServiceMode;
stSieve_Motor_Int.bCmdFwd R= _w7;
stSieve_Motor_Int.bCmdBwd R= _w7;
stSieve_Motor_Int.bCmdStop R= _w7;

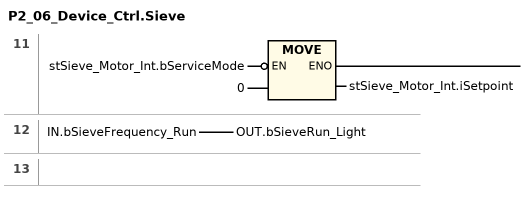
// NETWORK 11
IF NOT stSieve_Motor_Int.bServiceMode THEN stSieve_Motor_Int.iSetpoint := 0; END_IF

// NETWORK 12
OUT.bSieveRun_Light := IN.bSieveFrequency_Run;

// NETWORK 13
END_ACTION

ACTION SP_Mixer:
